Yaskawa INFORM job: pointsmerc3TRJ1.JBI

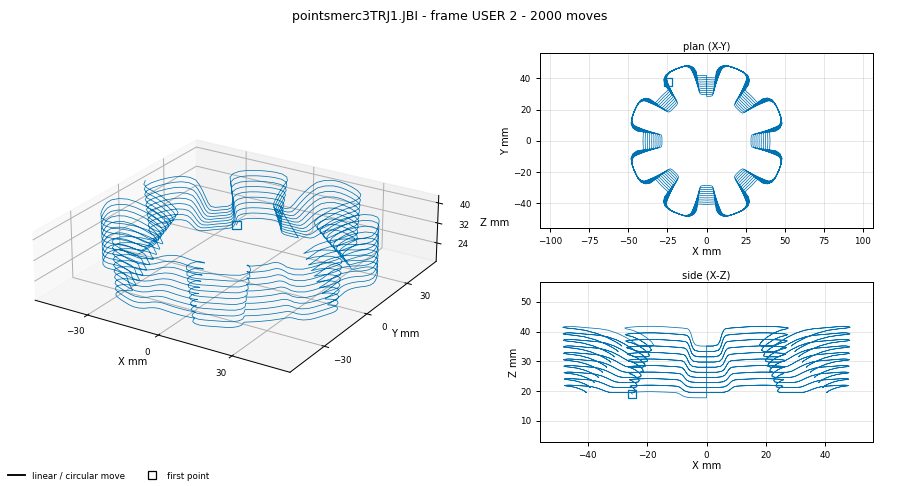
[picture p0: tool path of pointsmerc3TRJ1.JBI in frame USER 2, 2000 of 2000 moves have a stored position in this frame; points joined in program order, loops and branches not executed]
/JOB
//NAME pointsmerc3TRJ1
//POS
///NPOS 2000,0,0,0,0,0
///USER 2
///TOOL 1
///POSTYPE USER
///RECTAN
///RCONF 1,0,0,0,0,0,0,0,0,0,0,0,0,0,0,0,0,0,0,0,0,0,0,0
C00000=-24.917,37.674,19.017,179.9472,0.1674,0.0000
C00001=-25.352,39.110,19.349,-179.2805,-2.8495,0.0000
C00002=-25.558,40.564,19.514,179.7705,-3.0354,0.0000
C00003=-25.030,42.161,19.602,179.1176,-1.5538,0.0000
C00004=-23.802,43.680,19.673,179.0591,-0.8568,0.0000
C00005=-22.056,44.839,19.746,179.9560,-0.0226,0.0000
C00006=-20.124,45.768,19.794,179.9935,-0.0029,0.0000
C00007=-18.133,46.592,19.794,179.9934,-0.0025,0.0000
C00008=-16.110,47.302,19.746,179.9530,-0.0151,0.0000
C00009=-14.056,47.717,19.673,178.7288,-0.0593,0.0000
C00010=-12.113,47.511,19.602,178.2774,0.4749,0.0000
C00011=-10.611,46.755,19.514,177.6906,1.9837,0.0000
C00012=-9.729,45.582,19.349,178.4925,2.5230,0.0000
C00013=-9.020,44.258,19.017,-179.9189,-0.1557,0.0000
C00014=-8.331,43.070,18.587,-176.3263,-5.7834,0.0000
C00015=-7.515,42.203,18.169,-165.2639,-13.0795,0.0000
C00016=-6.279,41.769,17.866,-146.1512,-5.7263,0.0000
C00017=-4.265,41.794,17.745,-142.9346,1.8354,0.0000
C00018=-2.165,41.942,17.740,-142.7693,1.9023,0.0000
C00019=0.000,41.999,17.743,-142.7393,0.0003,0.0000
C00020=0.000,40.651,19.482,-141.7566,0.0003,0.0000
C00021=2.042,40.599,19.478,-141.7861,-1.9186,0.0000
C00022=4.057,40.463,19.484,-141.9733,-1.4629,0.0000
C00023=6.024,40.479,19.630,-146.2958,7.7682,0.0000
C00024=7.200,41.019,19.996,-169.0806,12.4470,0.0000
C00025=7.966,42.055,20.504,-178.0973,3.7099,0.0000
C00026=8.617,43.471,21.031,179.2926,-1.6631,0.0000
C00027=9.290,45.059,21.441,177.9597,-4.2609,0.0000
C00028=10.130,46.493,21.645,176.7689,-3.4833,0.0000
C00029=11.658,47.456,21.754,177.4448,-0.9082,0.0000
C00030=13.694,47.783,21.842,178.3657,0.0207,0.0000
C00031=15.881,47.377,21.932,179.9236,0.0242,0.0000
C00032=18.055,46.622,21.992,179.9901,0.0038,0.0000
C00033=20.200,45.734,21.992,179.9903,0.0044,0.0000
C00034=22.271,44.730,21.932,179.9289,0.0369,0.0000
C00035=24.104,43.471,21.842,178.8296,1.1409,0.0000
C00036=25.313,41.801,21.754,178.8351,2.4489,0.0000
C00037=25.713,40.038,21.645,-179.8172,4.7463,0.0000
C00038=25.293,38.430,21.441,-178.4233,4.4530,0.0000
C00039=24.645,36.832,21.031,-179.3238,1.6761,0.0000
C00040=24.105,35.370,20.504,178.7177,-3.9670,0.0000
C00041=23.913,34.096,19.996,178.7089,-16.4515,0.0000
C00042=24.363,32.883,19.630,-160.4193,-28.9701,0.0000
C00043=25.743,31.481,19.484,-150.0620,-24.6708,0.0000
C00044=27.264,30.151,19.478,-149.5929,-24.4247,0.0000
C00045=28.745,28.745,19.482,-150.8690,-25.9576,0.0000
C00046=30.151,27.264,19.478,-152.2298,-27.4413,0.0000
C00047=31.481,25.743,19.484,-152.0729,-26.9678,0.0000
C00048=32.883,24.363,19.630,-149.5613,-17.0504,0.0000
C00049=34.096,23.913,19.996,-163.5445,1.2382,0.0000
C00050=35.370,24.105,20.504,-176.0321,1.2792,0.0000
C00051=36.832,24.645,21.031,178.3238,-0.6759,0.0000
C00052=38.430,25.293,21.441,175.5453,-1.5719,0.0000
C00053=40.038,25.713,21.645,175.2537,-0.1822,0.0000
C00054=41.801,25.313,21.754,177.5506,1.1638,0.0000
C00055=43.471,24.104,21.842,178.8588,1.1702,0.0000
C00056=44.730,22.271,21.932,179.9631,0.0711,0.0000
C00057=45.734,20.200,21.992,179.9956,0.0097,0.0000
C00058=46.622,18.055,21.992,179.9962,0.0099,0.0000
C00059=47.377,15.881,21.932,179.9758,0.0764,0.0000
C00060=47.783,13.694,21.842,179.9793,1.6343,0.0000
C00061=47.456,11.658,21.754,-179.0909,2.5548,0.0000
C00062=46.493,10.130,21.645,-176.5112,3.2252,0.0000
C00063=45.059,9.290,21.441,-175.7364,2.0346,0.0000
C00064=43.471,8.617,21.031,-178.3368,0.7071,0.0000
C00065=42.055,7.966,20.504,176.2881,-1.8987,0.0000
C00066=41.019,7.200,19.996,167.3309,-10.6597,0.0000
C00067=40.479,6.024,19.630,170.6874,-33.3542,0.0000
C00068=40.463,4.057,19.484,-178.1431,-38.0121,0.0000
C00069=40.599,2.042,19.478,-177.5587,-38.1886,0.0000
C00070=40.651,0.000,19.482,179.9997,-38.2434,0.0000
C00071=40.599,-2.042,19.478,177.5592,-38.1887,0.0000
C00072=40.463,-4.057,19.484,178.1450,-38.0120,0.0000
C00073=40.479,-6.024,19.630,-170.6883,-33.3546,0.0000
C00074=41.019,-7.200,19.996,-167.3309,-10.6597,0.0000
C00075=42.055,-7.966,20.504,-176.2881,-1.8987,0.0000
C00076=43.471,-8.617,21.031,178.3368,0.7071,0.0000
C00077=45.059,-9.290,21.441,175.7364,2.0346,0.0000
C00078=46.493,-10.130,21.645,176.5112,3.2252,0.0000
C00079=47.456,-11.658,21.754,179.0909,2.5548,0.0000
C00080=47.783,-13.694,21.842,-179.9793,1.6343,0.0000
C00081=47.377,-15.881,21.932,-179.9758,0.0764,0.0000
C00082=46.622,-18.055,21.992,-179.9962,0.0099,0.0000
C00083=45.734,-20.200,21.992,-179.9956,0.0097,0.0000
C00084=44.730,-22.271,21.932,-179.9631,0.0711,0.0000
C00085=43.471,-24.104,21.842,-178.8588,1.1702,0.0000
C00086=41.801,-25.313,21.754,-177.5506,1.1638,0.0000
C00087=40.038,-25.713,21.645,-175.2537,-0.1822,0.0000
C00088=38.430,-25.293,21.441,-175.5453,-1.5719,0.0000
C00089=36.832,-24.645,21.031,-178.3238,-0.6759,0.0000
C00090=35.370,-24.105,20.504,176.0321,1.2792,0.0000
C00091=34.096,-23.913,19.996,163.5445,1.2382,0.0000
C00092=32.883,-24.363,19.630,149.5611,-17.0496,0.0000
C00093=31.481,-25.743,19.484,152.0737,-26.9690,0.0000
C00094=30.151,-27.264,19.478,152.2301,-27.4416,0.0000
C00095=28.745,-28.745,19.482,150.8686,-25.9571,0.0000
C00096=27.264,-30.151,19.478,149.5931,-24.4250,0.0000
C00097=25.743,-31.481,19.484,150.0631,-24.6718,0.0000
C00098=24.363,-32.883,19.630,160.4184,-28.9698,0.0000
C00099=23.913,-34.096,19.996,-178.7089,-16.4515,0.0000
C00100=24.105,-35.370,20.504,-178.7177,-3.9670,0.0000
C00101=24.645,-36.832,21.031,179.3238,1.6761,0.0000
C00102=25.293,-38.430,21.441,178.4233,4.4530,0.0000
C00103=25.713,-40.038,21.645,179.8172,4.7463,0.0000
C00104=25.313,-41.801,21.754,-178.8351,2.4489,0.0000
C00105=24.104,-43.471,21.842,-178.8296,1.1409,0.0000
C00106=22.271,-44.730,21.932,-179.9289,0.0369,0.0000
C00107=20.200,-45.734,21.992,-179.9903,0.0044,0.0000
C00108=18.055,-46.622,21.992,-179.9901,0.0038,0.0000
C00109=15.881,-47.377,21.932,-179.9236,0.0242,0.0000
C00110=13.694,-47.783,21.842,-178.3657,0.0207,0.0000
C00111=11.658,-47.456,21.754,-177.4448,-0.9082,0.0000
C00112=10.130,-46.493,21.645,-176.7689,-3.4833,0.0000
C00113=9.290,-45.059,21.441,-177.9597,-4.2609,0.0000
C00114=8.617,-43.471,21.031,-179.2926,-1.6631,0.0000
C00115=7.966,-42.055,20.504,178.0973,3.7099,0.0000
C00116=7.200,-41.019,19.996,169.0806,12.4470,0.0000
C00117=6.024,-40.479,19.630,146.2958,7.7682,0.0000
C00118=4.057,-40.463,19.484,141.9733,-1.4629,0.0000
C00119=2.042,-40.599,19.478,141.7861,-1.9186,0.0000
C00120=0.000,-40.651,19.482,141.7566,0.0003,0.0000
C00121=0.000,-40.651,19.482,141.7566,0.0003,0.0000
C00122=-2.042,-40.599,19.478,141.7861,1.9182,0.0000
C00123=-4.057,-40.463,19.484,141.9735,1.4614,0.0000
C00124=-6.024,-40.479,19.630,146.2954,-7.7675,0.0000
C00125=-7.200,-41.019,19.996,169.0806,-12.4470,0.0000
C00126=-7.966,-42.055,20.504,178.0973,-3.7099,0.0000
C00127=-8.617,-43.471,21.031,-179.2926,1.6631,0.0000
C00128=-9.290,-45.059,21.441,-177.9597,4.2609,0.0000
C00129=-10.130,-46.493,21.645,-176.7689,3.4833,0.0000
C00130=-11.658,-47.456,21.754,-177.4448,0.9082,0.0000
C00131=-13.694,-47.783,21.842,-178.3657,-0.0207,0.0000
C00132=-15.881,-47.377,21.932,-179.9236,-0.0242,0.0000
C00133=-18.055,-46.622,21.992,-179.9901,-0.0038,0.0000
C00134=-20.200,-45.734,21.992,-179.9903,-0.0044,0.0000
C00135=-22.271,-44.730,21.932,-179.9289,-0.0369,0.0000
C00136=-24.104,-43.471,21.842,-178.8296,-1.1409,0.0000
C00137=-25.313,-41.801,21.754,-178.8351,-2.4489,0.0000
C00138=-25.713,-40.038,21.645,179.8172,-4.7463,0.0000
C00139=-25.293,-38.430,21.441,178.4233,-4.4530,0.0000
C00140=-24.645,-36.832,21.031,179.3238,-1.6761,0.0000
C00141=-24.105,-35.370,20.504,-178.7177,3.9670,0.0000
C00142=-23.913,-34.096,19.996,-178.7089,16.4515,0.0000
C00143=-24.363,-32.883,19.630,160.4193,28.9701,0.0000
C00144=-25.743,-31.481,19.484,150.0620,24.6708,0.0000
C00145=-27.264,-30.151,19.478,149.5929,24.4247,0.0000
C00146=-28.745,-28.745,19.482,150.8690,25.9576,0.0000
C00147=-30.151,-27.264,19.478,152.2298,27.4413,0.0000
C00148=-31.481,-25.743,19.484,152.0729,26.9678,0.0000
C00149=-32.883,-24.363,19.630,149.5613,17.0504,0.0000
C00150=-34.096,-23.913,19.996,163.5445,-1.2382,0.0000
C00151=-35.370,-24.105,20.504,176.0321,-1.2792,0.0000
C00152=-36.832,-24.645,21.031,-178.3238,0.6759,0.0000
C00153=-38.430,-25.293,21.441,-175.5453,1.5719,0.0000
C00154=-40.038,-25.713,21.645,-175.2537,0.1822,0.0000
C00155=-41.801,-25.313,21.754,-177.5506,-1.1638,0.0000
C00156=-43.471,-24.104,21.842,-178.8588,-1.1702,0.0000
C00157=-44.730,-22.271,21.932,-179.9631,-0.0711,0.0000
C00158=-45.734,-20.200,21.992,-179.9956,-0.0097,0.0000
C00159=-46.622,-18.055,21.992,-179.9962,-0.0099,0.0000
C00160=-47.377,-15.881,21.932,-179.9758,-0.0764,0.0000
C00161=-47.783,-13.694,21.842,-179.9793,-1.6343,0.0000
C00162=-47.456,-11.658,21.754,179.0909,-2.5548,0.0000
C00163=-46.493,-10.130,21.645,176.5112,-3.2252,0.0000
C00164=-45.059,-9.290,21.441,175.7364,-2.0346,0.0000
C00165=-43.471,-8.617,21.031,178.3368,-0.7071,0.0000
C00166=-42.055,-7.966,20.504,-176.2881,1.8987,0.0000
C00167=-41.019,-7.200,19.996,-167.3309,10.6597,0.0000
C00168=-40.479,-6.024,19.630,-170.6874,33.3542,0.0000
C00169=-40.463,-4.057,19.484,178.1431,38.0121,0.0000
C00170=-40.599,-2.042,19.478,177.5587,38.1886,0.0000
C00171=-40.651,0.000,19.482,-179.9997,38.2434,0.0000
C00172=-40.599,2.042,19.478,-177.5592,38.1887,0.0000
C00173=-40.463,4.057,19.484,-178.1450,38.0120,0.0000
C00174=-40.479,6.024,19.630,170.6883,33.3546,0.0000
C00175=-41.019,7.200,19.996,167.3309,10.6597,0.0000
C00176=-42.055,7.966,20.504,176.2881,1.8987,0.0000
C00177=-43.471,8.617,21.031,-178.3368,-0.7071,0.0000
C00178=-45.059,9.290,21.441,-175.7364,-2.0346,0.0000
C00179=-46.493,10.130,21.645,-176.5112,-3.2252,0.0000
C00180=-47.456,11.658,21.754,-179.0909,-2.5548,0.0000
C00181=-47.783,13.694,21.842,179.9793,-1.6343,0.0000
C00182=-47.377,15.881,21.932,179.9758,-0.0764,0.0000
C00183=-46.622,18.055,21.992,179.9962,-0.0099,0.0000
C00184=-45.734,20.200,21.992,179.9956,-0.0097,0.0000
C00185=-44.730,22.271,21.932,179.9631,-0.0711,0.0000
C00186=-43.471,24.104,21.842,178.8588,-1.1702,0.0000
C00187=-41.801,25.313,21.754,177.5506,-1.1638,0.0000
C00188=-40.038,25.713,21.645,175.2537,0.1822,0.0000
C00189=-38.430,25.293,21.441,175.5453,1.5719,0.0000
C00190=-36.832,24.645,21.031,178.3238,0.6759,0.0000
C00191=-35.370,24.105,20.504,-176.0321,-1.2792,0.0000
C00192=-34.096,23.913,19.996,-163.5445,-1.2382,0.0000
C00193=-32.883,24.363,19.630,-149.5611,17.0496,0.0000
C00194=-31.481,25.743,19.484,-152.0737,26.9690,0.0000
C00195=-30.151,27.264,19.478,-152.2301,27.4416,0.0000
C00196=-28.745,28.745,19.482,-150.8686,25.9571,0.0000
C00197=-27.264,30.151,19.478,-149.5931,24.4250,0.0000
C00198=-25.743,31.481,19.484,-150.0631,24.6718,0.0000
C00199=-24.363,32.883,19.630,-160.4184,28.9698,0.0000
C00200=-23.913,34.096,19.996,178.7089,16.4515,0.0000
C00201=-24.105,35.370,20.504,178.7177,3.9670,0.0000
C00202=-24.645,36.832,21.031,-179.3238,-1.6761,0.0000
C00203=-25.293,38.430,21.441,-178.4233,-4.4530,0.0000
C00204=-25.713,40.038,21.645,-179.8172,-4.7463,0.0000
C00205=-25.313,41.801,21.754,178.8351,-2.4489,0.0000
C00206=-24.104,43.471,21.842,178.8296,-1.1409,0.0000
C00207=-22.271,44.730,21.932,179.9289,-0.0369,0.0000
C00208=-20.200,45.734,21.992,179.9903,-0.0044,0.0000
C00209=-18.055,46.622,21.992,179.9901,-0.0038,0.0000
C00210=-15.881,47.377,21.932,179.9236,-0.0242,0.0000
C00211=-13.694,47.783,21.842,178.3657,-0.0207,0.0000
C00212=-11.658,47.456,21.754,177.4448,0.9082,0.0000
C00213=-10.130,46.493,21.645,176.7689,3.4833,0.0000
C00214=-9.290,45.059,21.441,177.9597,4.2609,0.0000
C00215=-8.617,43.471,21.031,179.2926,1.6631,0.0000
C00216=-7.966,42.055,20.504,-178.0973,-3.7099,0.0000
C00217=-7.200,41.019,19.996,-169.0806,-12.4470,0.0000
C00218=-6.024,40.479,19.630,-146.2954,-7.7675,0.0000
C00219=-4.057,40.463,19.484,-141.9735,1.4614,0.0000
C00220=-2.042,40.599,19.478,-141.7861,1.9182,0.0000
C00221=0.000,40.651,19.482,-141.7566,0.0003,0.0000
C00222=0.000,39.279,21.202,-141.1100,0.0002,0.0000
C00223=1.916,39.231,21.197,-141.1387,-1.9150,0.0000
C00224=3.846,39.107,21.204,-141.3582,-1.0288,0.0000
C00225=5.765,39.166,21.375,-147.0450,9.7425,0.0000
C00226=6.881,39.812,21.808,-172.3813,10.8619,0.0000
C00227=7.594,41.021,22.410,-179.2636,1.7324,0.0000
C00228=8.207,42.669,23.038,178.8678,-3.1758,0.0000
C00229=8.843,44.528,23.528,177.7717,-5.6527,0.0000
C00230=9.641,46.227,23.773,176.2825,-4.8520,0.0000
C00231=11.196,47.401,23.904,176.7678,-1.3919,0.0000
C00232=13.327,47.850,24.010,178.0518,-0.0356,0.0000
C00233=15.648,47.454,24.119,179.8977,0.0319,0.0000
C00234=17.976,46.653,24.190,179.9872,0.0049,0.0000
C00235=20.278,45.699,24.190,179.9875,0.0056,0.0000
C00236=22.491,44.620,24.119,179.9051,0.0498,0.0000
C00237=24.412,43.258,24.010,178.6473,1.4026,0.0000
C00238=25.601,41.434,23.904,178.6983,3.2695,0.0000
C00239=25.871,39.504,23.773,-179.1860,6.0555,0.0000
C00240=25.233,37.739,23.528,-177.5648,5.5670,0.0000
C00241=24.369,35.974,23.038,-178.5526,3.0452,0.0000
C00242=23.637,34.376,22.410,179.2953,-1.7456,0.0000
C00243=23.286,33.017,21.808,177.5775,-13.0215,0.0000
C00244=23.618,31.771,21.375,-162.5821,-29.9181,0.0000
C00245=24.933,30.373,21.204,-149.8186,-25.3906,0.0000
C00246=26.385,29.096,21.197,-149.0304,-24.8212,0.0000
C00247=27.774,27.774,21.202,-150.3014,-26.3558,0.0000
C00248=29.096,26.385,21.197,-151.6568,-27.8426,0.0000
C00249=30.373,24.933,21.204,-151.2294,-27.0106,0.0000
C00250=31.771,23.618,21.375,-148.9059,-15.0382,0.0000
C00251=33.017,23.286,21.808,-166.9673,2.3601,0.0000
C00252=34.376,23.637,22.410,-178.2543,0.7044,0.0000
C00253=35.974,24.369,23.038,176.9538,-1.4453,0.0000
C00254=37.739,25.233,23.528,174.4280,-2.4237,0.0000
C00255=39.504,25.871,23.773,173.9439,-0.8094,0.0000
C00256=41.434,25.601,23.904,176.7297,1.2996,0.0000
C00257=43.258,24.412,24.010,178.5970,1.3523,0.0000
C00258=44.620,22.491,24.119,179.9502,0.0949,0.0000
C00259=45.699,20.278,24.190,179.9944,0.0125,0.0000
C00260=46.653,17.976,24.190,179.9951,0.0128,0.0000
C00261=47.454,15.648,24.119,179.9681,0.1023,0.0000
C00262=47.850,13.327,24.010,-179.9644,1.9482,0.0000
C00263=47.401,11.196,23.904,-178.6059,3.2312,0.0000
C00264=46.227,9.641,23.773,-175.1378,3.7041,0.0000
C00265=44.528,8.843,23.528,-174.3430,2.2175,0.0000
C00266=42.669,8.207,23.038,-176.8236,1.1304,0.0000
C00267=41.021,7.594,22.410,178.2674,-0.7361,0.0000
C00268=39.812,6.881,21.808,169.0437,-7.4814,0.0000
C00269=39.166,5.765,21.375,168.4358,-32.4210,0.0000
C00270=39.107,3.846,21.204,-178.6830,-38.6345,0.0000
C00271=39.231,1.916,21.197,-177.5412,-38.8355,0.0000
C00272=39.279,0.000,21.202,179.9998,-38.8900,0.0000
C00273=39.231,-1.916,21.197,177.5416,-38.8356,0.0000
C00274=39.107,-3.847,21.204,178.6850,-38.6342,0.0000
C00275=39.166,-5.765,21.375,-168.4365,-32.4215,0.0000
C00276=39.812,-6.881,21.808,-169.0437,-7.4814,0.0000
C00277=41.021,-7.594,22.410,-178.2674,-0.7361,0.0000
C00278=42.669,-8.207,23.038,176.8236,1.1304,0.0000
C00279=44.528,-8.843,23.528,174.3430,2.2175,0.0000
C00280=46.227,-9.641,23.773,175.1378,3.7041,0.0000
C00281=47.401,-11.196,23.904,178.6059,3.2312,0.0000
C00282=47.850,-13.327,24.010,179.9644,1.9482,0.0000
C00283=47.454,-15.648,24.119,-179.9681,0.1023,0.0000
C00284=46.653,-17.976,24.190,-179.9951,0.0128,0.0000
C00285=45.699,-20.278,24.190,-179.9944,0.0125,0.0000
C00286=44.620,-22.491,24.119,-179.9502,0.0949,0.0000
C00287=43.258,-24.412,24.010,-178.5970,1.3523,0.0000
C00288=41.434,-25.601,23.904,-176.7297,1.2996,0.0000
C00289=39.504,-25.871,23.773,-173.9439,-0.8094,0.0000
C00290=37.739,-25.233,23.528,-174.4280,-2.4237,0.0000
C00291=35.974,-24.369,23.038,-176.9538,-1.4453,0.0000
C00292=34.376,-23.637,22.410,178.2543,0.7044,0.0000
C00293=33.017,-23.286,21.808,166.9673,2.3601,0.0000
C00294=31.771,-23.618,21.375,148.9058,-15.0373,0.0000
C00295=30.373,-24.933,21.204,151.2304,-27.0120,0.0000
C00296=29.096,-26.385,21.197,151.6570,-27.8428,0.0000
C00297=27.774,-27.774,21.202,150.3012,-26.3555,0.0000
C00298=26.385,-29.096,21.197,149.0306,-24.8215,0.0000
C00299=24.933,-30.373,21.204,149.8199,-25.3917,0.0000
C00300=23.618,-31.771,21.375,162.5812,-29.9179,0.0000
C00301=23.286,-33.017,21.808,-177.5775,-13.0215,0.0000
C00302=23.637,-34.376,22.410,-179.2953,-1.7456,0.0000
C00303=24.369,-35.974,23.038,178.5526,3.0452,0.0000
C00304=25.233,-37.739,23.528,177.5648,5.5670,0.0000
C00305=25.871,-39.504,23.773,179.1860,6.0555,0.0000
C00306=25.601,-41.434,23.904,-178.6983,3.2695,0.0000
C00307=24.412,-43.258,24.010,-178.6473,1.4026,0.0000
C00308=22.491,-44.620,24.119,-179.9051,0.0498,0.0000
C00309=20.278,-45.699,24.190,-179.9875,0.0056,0.0000
C00310=17.976,-46.653,24.190,-179.9872,0.0049,0.0000
C00311=15.648,-47.454,24.119,-179.8977,0.0319,0.0000
C00312=13.327,-47.850,24.010,-178.0518,-0.0356,0.0000
C00313=11.196,-47.401,23.904,-176.7678,-1.3919,0.0000
C00314=9.641,-46.227,23.773,-176.2825,-4.8520,0.0000
C00315=8.843,-44.528,23.528,-177.7717,-5.6527,0.0000
C00316=8.207,-42.669,23.038,-178.8678,-3.1758,0.0000
C00317=7.594,-41.021,22.410,179.2636,1.7324,0.0000
C00318=6.881,-39.812,21.808,172.3813,10.8619,0.0000
C00319=5.765,-39.166,21.375,147.0450,9.7425,0.0000
C00320=3.846,-39.107,21.204,141.3582,-1.0288,0.0000
C00321=1.916,-39.231,21.197,141.1387,-1.9150,0.0000
C00322=0.000,-39.279,21.202,141.1100,0.0002,0.0000
C00323=0.000,-39.279,21.202,141.1100,0.0002,0.0000
C00324=-1.916,-39.231,21.197,141.1386,1.9147,0.0000
C00325=-3.847,-39.107,21.204,141.3584,1.0272,0.0000
C00326=-5.765,-39.166,21.375,147.0445,-9.7418,0.0000
C00327=-6.881,-39.812,21.808,172.3813,-10.8619,0.0000
C00328=-7.594,-41.021,22.410,179.2636,-1.7324,0.0000
C00329=-8.207,-42.669,23.038,-178.8678,3.1758,0.0000
C00330=-8.843,-44.528,23.528,-177.7717,5.6527,0.0000
C00331=-9.641,-46.227,23.773,-176.2825,4.8520,0.0000
C00332=-11.196,-47.401,23.904,-176.7678,1.3919,0.0000
C00333=-13.327,-47.850,24.010,-178.0518,0.0356,0.0000
C00334=-15.648,-47.454,24.119,-179.8977,-0.0319,0.0000
C00335=-17.976,-46.653,24.190,-179.9872,-0.0049,0.0000
C00336=-20.278,-45.699,24.190,-179.9875,-0.0056,0.0000
C00337=-22.491,-44.620,24.119,-179.9051,-0.0498,0.0000
C00338=-24.412,-43.258,24.010,-178.6473,-1.4026,0.0000
C00339=-25.601,-41.434,23.904,-178.6983,-3.2695,0.0000
C00340=-25.871,-39.504,23.773,179.1860,-6.0555,0.0000
C00341=-25.233,-37.739,23.528,177.5648,-5.5670,0.0000
C00342=-24.369,-35.974,23.038,178.5526,-3.0452,0.0000
C00343=-23.637,-34.376,22.410,-179.2953,1.7456,0.0000
C00344=-23.286,-33.017,21.808,-177.5775,13.0215,0.0000
C00345=-23.618,-31.771,21.375,162.5821,29.9181,0.0000
C00346=-24.933,-30.373,21.204,149.8186,25.3906,0.0000
C00347=-26.385,-29.096,21.197,149.0304,24.8212,0.0000
C00348=-27.774,-27.774,21.202,150.3014,26.3558,0.0000
C00349=-29.096,-26.385,21.197,151.6568,27.8426,0.0000
C00350=-30.373,-24.933,21.204,151.2294,27.0106,0.0000
C00351=-31.771,-23.618,21.375,148.9059,15.0382,0.0000
C00352=-33.017,-23.286,21.808,166.9673,-2.3601,0.0000
C00353=-34.376,-23.637,22.410,178.2543,-0.7044,0.0000
C00354=-35.974,-24.369,23.038,-176.9538,1.4453,0.0000
C00355=-37.739,-25.233,23.528,-174.4280,2.4237,0.0000
C00356=-39.504,-25.871,23.773,-173.9439,0.8094,0.0000
C00357=-41.434,-25.601,23.904,-176.7297,-1.2996,0.0000
C00358=-43.258,-24.412,24.010,-178.5970,-1.3523,0.0000
C00359=-44.620,-22.491,24.119,-179.9502,-0.0949,0.0000
C00360=-45.699,-20.278,24.190,-179.9944,-0.0125,0.0000
C00361=-46.653,-17.976,24.190,-179.9951,-0.0128,0.0000
C00362=-47.454,-15.648,24.119,-179.9681,-0.1023,0.0000
C00363=-47.850,-13.327,24.010,179.9644,-1.9482,0.0000
C00364=-47.401,-11.196,23.904,178.6059,-3.2312,0.0000
C00365=-46.227,-9.641,23.773,175.1378,-3.7041,0.0000
C00366=-44.528,-8.843,23.528,174.3430,-2.2175,0.0000
C00367=-42.669,-8.207,23.038,176.8236,-1.1304,0.0000
C00368=-41.021,-7.594,22.410,-178.2674,0.7361,0.0000
C00369=-39.812,-6.881,21.808,-169.0437,7.4814,0.0000
C00370=-39.166,-5.765,21.375,-168.4358,32.4210,0.0000
C00371=-39.107,-3.846,21.204,178.6830,38.6345,0.0000
C00372=-39.231,-1.916,21.197,177.5412,38.8355,0.0000
C00373=-39.279,0.000,21.202,-179.9998,38.8900,0.0000
C00374=-39.231,1.916,21.197,-177.5416,38.8356,0.0000
C00375=-39.107,3.847,21.204,-178.6850,38.6342,0.0000
C00376=-39.166,5.765,21.375,168.4365,32.4215,0.0000
C00377=-39.812,6.881,21.808,169.0437,7.4814,0.0000
C00378=-41.021,7.594,22.410,178.2674,0.7361,0.0000
C00379=-42.669,8.207,23.038,-176.8236,-1.1304,0.0000
C00380=-44.528,8.843,23.528,-174.3430,-2.2175,0.0000
C00381=-46.227,9.641,23.773,-175.1378,-3.7041,0.0000
C00382=-47.401,11.196,23.904,-178.6059,-3.2312,0.0000
C00383=-47.850,13.327,24.010,-179.9644,-1.9482,0.0000
C00384=-47.454,15.648,24.119,179.9681,-0.1023,0.0000
C00385=-46.653,17.976,24.190,179.9951,-0.0128,0.0000
C00386=-45.699,20.278,24.190,179.9944,-0.0125,0.0000
C00387=-44.620,22.491,24.119,179.9502,-0.0949,0.0000
C00388=-43.258,24.412,24.010,178.5970,-1.3523,0.0000
C00389=-41.434,25.601,23.904,176.7297,-1.2996,0.0000
C00390=-39.504,25.871,23.773,173.9439,0.8094,0.0000
C00391=-37.739,25.233,23.528,174.4280,2.4237,0.0000
C00392=-35.974,24.369,23.038,176.9538,1.4453,0.0000
C00393=-34.376,23.637,22.410,-178.2543,-0.7044,0.0000
C00394=-33.017,23.286,21.808,-166.9673,-2.3601,0.0000
C00395=-31.771,23.618,21.375,-148.9058,15.0373,0.0000
C00396=-30.373,24.933,21.204,-151.2304,27.0120,0.0000
C00397=-29.096,26.385,21.197,-151.6570,27.8428,0.0000
C00398=-27.774,27.774,21.202,-150.3012,26.3555,0.0000
C00399=-26.385,29.096,21.197,-149.0306,24.8215,0.0000
C00400=-24.933,30.373,21.204,-149.8199,25.3917,0.0000
C00401=-23.618,31.771,21.375,-162.5812,29.9179,0.0000
C00402=-23.286,33.017,21.808,177.5775,13.0215,0.0000
C00403=-23.637,34.376,22.410,179.2953,1.7456,0.0000
C00404=-24.369,35.974,23.038,-178.5526,-3.0452,0.0000
C00405=-25.233,37.739,23.528,-177.5648,-5.5670,0.0000
C00406=-25.871,39.504,23.773,-179.1860,-6.0555,0.0000
C00407=-25.601,41.434,23.904,178.6983,-3.2695,0.0000
C00408=-24.412,43.258,24.010,178.6473,-1.4026,0.0000
C00409=-22.491,44.620,24.119,179.9051,-0.0498,0.0000
C00410=-20.278,45.699,24.190,179.9875,-0.0056,0.0000
C00411=-17.976,46.653,24.190,179.9872,-0.0049,0.0000
C00412=-15.648,47.454,24.119,179.8977,-0.0319,0.0000
C00413=-13.327,47.850,24.010,178.0518,0.0356,0.0000
C00414=-11.196,47.401,23.904,176.7678,1.3919,0.0000
C00415=-9.641,46.227,23.773,176.2825,4.8520,0.0000
C00416=-8.843,44.528,23.528,177.7717,5.6527,0.0000
C00417=-8.207,42.669,23.038,178.8678,3.1758,0.0000
C00418=-7.594,41.021,22.410,-179.2636,-1.7324,0.0000
C00419=-6.881,39.812,21.808,-172.3813,-10.8619,0.0000
C00420=-5.765,39.166,21.375,-147.0445,-9.7418,0.0000
C00421=-3.847,39.107,21.204,-141.3584,1.0272,0.0000
C00422=-1.916,39.231,21.197,-141.1386,1.9147,0.0000
C00423=0.000,39.279,21.202,-141.1100,0.0002,0.0000
C00424=0.000,37.892,22.909,-140.7729,0.0001,0.0000
C00425=1.790,37.849,22.904,-140.8005,-1.8934,0.0000
C00426=3.633,37.737,22.912,-141.0647,-0.5438,0.0000
C00427=5.504,37.838,23.110,-148.3550,11.5394,0.0000
C00428=6.557,38.594,23.612,-174.9776,8.7701,0.0000
C00429=7.219,39.979,24.311,-179.9995,0.0014,0.0000
C00430=7.794,41.862,25.043,178.6707,-4.3586,0.0000
C00431=8.395,43.994,25.615,177.7869,-6.6761,0.0000
C00432=9.151,45.960,25.902,176.1277,-5.9542,0.0000
C00433=10.734,47.345,26.054,176.2738,-1.8650,0.0000
C00434=12.959,47.917,26.178,177.8036,-0.1012,0.0000
C00435=15.415,47.531,26.305,179.8764,0.0380,0.0000
C00436=17.897,46.683,26.389,179.9849,0.0057,0.0000
C00437=20.355,45.665,26.389,179.9853,0.0067,0.0000
C00438=22.710,44.510,26.305,179.8857,0.0605,0.0000
C00439=24.719,43.046,26.178,178.5181,1.6245,0.0000
C00440=25.888,41.068,26.054,178.6837,3.9532,0.0000
C00441=26.028,38.969,25.902,-178.5075,6.9409,0.0000
C00442=25.172,37.045,25.615,-176.8232,6.2765,0.0000
C00443=24.090,35.112,25.043,-177.8523,4.0195,0.0000
C00444=23.165,33.374,24.311,179.9993,-0.0014,0.0000
C00445=22.654,31.927,23.612,177.2881,-9.7292,0.0000
C00446=22.864,30.647,23.110,-165.0937,-30.3273,0.0000
C00447=24.115,29.253,22.912,-149.8901,-25.9537,0.0000
C00448=25.498,28.029,22.904,-148.7483,-25.0431,0.0000
C00449=26.793,26.793,22.909,-150.0040,-26.5624,0.0000
C00450=28.029,25.498,22.904,-151.3420,-28.0359,0.0000
C00451=29.253,24.115,22.912,-150.6345,-26.8106,0.0000
C00452=30.647,22.864,23.110,-148.8108,-12.8294,0.0000
C00453=31.927,22.654,23.612,-170.2601,2.6728,0.0000
C00454=33.374,23.165,24.311,-179.9986,0.0007,0.0000
C00455=35.112,24.090,25.043,175.9777,-2.1424,0.0000
C00456=37.045,25.172,25.615,173.7139,-3.1578,0.0000
C00457=38.969,26.028,25.902,173.0567,-1.4816,0.0000
C00458=41.068,25.888,26.054,176.0457,1.3131,0.0000
C00459=43.046,24.719,26.178,178.3750,1.4813,0.0000
C00460=44.510,22.710,26.305,179.9395,0.1143,0.0000
C00461=45.665,20.355,26.389,179.9933,0.0147,0.0000
C00462=46.683,17.897,26.389,179.9943,0.0151,0.0000
C00463=47.531,15.415,26.305,179.9620,0.1236,0.0000
C00464=47.917,12.959,26.178,-179.8987,2.1964,0.0000
C00465=47.345,10.734,26.054,-178.1310,3.7242,0.0000
C00466=45.960,9.151,25.902,-174.0323,3.8514,0.0000
C00467=43.994,8.395,25.615,-173.3189,2.1980,0.0000
C00468=41.862,7.794,25.043,-175.6402,1.3254,0.0000
C00469=39.979,7.219,24.311,179.9986,-0.0005,0.0000
C00470=38.594,6.557,23.612,171.1966,-4.9635,0.0000
C00471=37.838,5.504,23.110,166.5136,-30.9339,0.0000
C00472=37.737,3.633,22.912,-179.3009,-38.9332,0.0000
C00473=37.849,1.790,22.904,-177.5573,-39.1740,0.0000
C00474=37.892,0.000,22.909,179.9999,-39.2271,0.0000
C00475=37.849,-1.790,22.904,177.5576,-39.1740,0.0000
C00476=37.737,-3.633,22.912,179.3032,-38.9330,0.0000
C00477=37.838,-5.504,23.110,-166.5142,-30.9345,0.0000
C00478=38.594,-6.557,23.612,-171.1966,-4.9635,0.0000
C00479=39.979,-7.219,24.311,-179.9986,-0.0005,0.0000
C00480=41.862,-7.794,25.043,175.6402,1.3254,0.0000
C00481=43.994,-8.395,25.615,173.3189,2.1980,0.0000
C00482=45.960,-9.151,25.902,174.0323,3.8514,0.0000
C00483=47.345,-10.734,26.054,178.1310,3.7242,0.0000
C00484=47.917,-12.959,26.178,179.8987,2.1964,0.0000
C00485=47.531,-15.415,26.305,-179.9620,0.1236,0.0000
C00486=46.683,-17.897,26.389,-179.9943,0.0151,0.0000
C00487=45.665,-20.355,26.389,-179.9933,0.0147,0.0000
C00488=44.510,-22.710,26.305,-179.9395,0.1143,0.0000
C00489=43.046,-24.719,26.178,-178.3750,1.4813,0.0000
C00490=41.068,-25.888,26.054,-176.0457,1.3131,0.0000
C00491=38.969,-26.028,25.902,-173.0567,-1.4816,0.0000
C00492=37.045,-25.172,25.615,-173.7139,-3.1578,0.0000
C00493=35.112,-24.090,25.043,-175.9777,-2.1424,0.0000
C00494=33.374,-23.165,24.311,179.9986,0.0007,0.0000
C00495=31.927,-22.654,23.612,170.2601,2.6728,0.0000
C00496=30.647,-22.864,23.110,148.8108,-12.8287,0.0000
C00497=29.253,-24.115,22.912,150.6355,-26.8122,0.0000
C00498=28.029,-25.498,22.904,151.3422,-28.0360,0.0000
C00499=26.793,-26.793,22.909,150.0039,-26.5623,0.0000
C00500=25.498,-28.029,22.904,148.7484,-25.0433,0.0000
C00501=24.115,-29.253,22.912,149.8915,-25.9549,0.0000
C00502=22.864,-30.647,23.110,165.0929,-30.3272,0.0000
C00503=22.654,-31.927,23.612,-177.2881,-9.7292,0.0000
C00504=23.165,-33.374,24.311,-179.9993,-0.0014,0.0000
C00505=24.090,-35.112,25.043,177.8523,4.0195,0.0000
C00506=25.172,-37.045,25.615,176.8232,6.2765,0.0000
C00507=26.028,-38.969,25.902,178.5075,6.9409,0.0000
C00508=25.888,-41.068,26.054,-178.6837,3.9532,0.0000
C00509=24.719,-43.046,26.178,-178.5181,1.6245,0.0000
C00510=22.710,-44.510,26.305,-179.8857,0.0605,0.0000
C00511=20.355,-45.665,26.389,-179.9853,0.0067,0.0000
C00512=17.897,-46.683,26.389,-179.9849,0.0057,0.0000
C00513=15.415,-47.531,26.305,-179.8764,0.0380,0.0000
C00514=12.959,-47.917,26.178,-177.8036,-0.1012,0.0000
C00515=10.734,-47.345,26.054,-176.2738,-1.8650,0.0000
C00516=9.151,-45.960,25.902,-176.1277,-5.9542,0.0000
C00517=8.395,-43.994,25.615,-177.7869,-6.6761,0.0000
C00518=7.794,-41.862,25.043,-178.6707,-4.3586,0.0000
C00519=7.219,-39.979,24.311,179.9995,0.0014,0.0000
C00520=6.557,-38.594,23.612,174.9776,8.7701,0.0000
C00521=5.504,-37.838,23.110,148.3550,11.5394,0.0000
C00522=3.633,-37.737,22.912,141.0647,-0.5438,0.0000
C00523=1.790,-37.849,22.904,140.8005,-1.8934,0.0000
C00524=0.000,-37.892,22.909,140.7729,0.0001,0.0000
C00525=0.000,-37.892,22.909,140.7729,0.0001,0.0000
C00526=-1.790,-37.849,22.904,140.8005,1.8932,0.0000
C00527=-3.633,-37.737,22.912,141.0650,0.5420,0.0000
C00528=-5.504,-37.838,23.110,148.3545,-11.5388,0.0000
C00529=-6.557,-38.594,23.612,174.9776,-8.7701,0.0000
C00530=-7.219,-39.979,24.311,179.9995,-0.0014,0.0000
C00531=-7.794,-41.862,25.043,-178.6707,4.3586,0.0000
C00532=-8.395,-43.994,25.615,-177.7869,6.6761,0.0000
C00533=-9.151,-45.960,25.902,-176.1277,5.9542,0.0000
C00534=-10.734,-47.345,26.054,-176.2738,1.8650,0.0000
C00535=-12.959,-47.917,26.178,-177.8036,0.1012,0.0000
C00536=-15.415,-47.531,26.305,-179.8764,-0.0380,0.0000
C00537=-17.897,-46.683,26.389,-179.9849,-0.0057,0.0000
C00538=-20.355,-45.665,26.389,-179.9853,-0.0067,0.0000
C00539=-22.710,-44.510,26.305,-179.8857,-0.0605,0.0000
C00540=-24.719,-43.046,26.178,-178.5181,-1.6245,0.0000
C00541=-25.888,-41.068,26.054,-178.6837,-3.9532,0.0000
C00542=-26.028,-38.969,25.902,178.5075,-6.9409,0.0000
C00543=-25.172,-37.045,25.615,176.8232,-6.2765,0.0000
C00544=-24.090,-35.112,25.043,177.8523,-4.0195,0.0000
C00545=-23.165,-33.374,24.311,-179.9993,0.0014,0.0000
C00546=-22.654,-31.927,23.612,-177.2881,9.7292,0.0000
C00547=-22.864,-30.647,23.110,165.0937,30.3273,0.0000
C00548=-24.115,-29.253,22.912,149.8901,25.9537,0.0000
C00549=-25.498,-28.029,22.904,148.7483,25.0431,0.0000
C00550=-26.793,-26.793,22.909,150.0040,26.5624,0.0000
C00551=-28.029,-25.498,22.904,151.3420,28.0359,0.0000
C00552=-29.253,-24.115,22.912,150.6345,26.8106,0.0000
C00553=-30.647,-22.864,23.110,148.8108,12.8294,0.0000
C00554=-31.927,-22.654,23.612,170.2601,-2.6728,0.0000
C00555=-33.374,-23.165,24.311,179.9986,-0.0007,0.0000
C00556=-35.112,-24.090,25.043,-175.9777,2.1424,0.0000
C00557=-37.045,-25.172,25.615,-173.7139,3.1578,0.0000
C00558=-38.969,-26.028,25.902,-173.0567,1.4816,0.0000
C00559=-41.068,-25.888,26.054,-176.0457,-1.3131,0.0000
C00560=-43.046,-24.719,26.178,-178.3750,-1.4813,0.0000
C00561=-44.510,-22.710,26.305,-179.9395,-0.1143,0.0000
C00562=-45.665,-20.355,26.389,-179.9933,-0.0147,0.0000
C00563=-46.683,-17.897,26.389,-179.9943,-0.0151,0.0000
C00564=-47.531,-15.415,26.305,-179.9620,-0.1236,0.0000
C00565=-47.917,-12.959,26.178,179.8987,-2.1964,0.0000
C00566=-47.345,-10.734,26.054,178.1310,-3.7242,0.0000
C00567=-45.960,-9.151,25.902,174.0323,-3.8514,0.0000
C00568=-43.994,-8.395,25.615,173.3189,-2.1980,0.0000
C00569=-41.862,-7.794,25.043,175.6402,-1.3254,0.0000
C00570=-39.979,-7.219,24.311,-179.9986,0.0005,0.0000
C00571=-38.594,-6.557,23.612,-171.1966,4.9635,0.0000
C00572=-37.838,-5.504,23.110,-166.5136,30.9339,0.0000
C00573=-37.737,-3.633,22.912,179.3009,38.9332,0.0000
C00574=-37.849,-1.790,22.904,177.5573,39.1740,0.0000
C00575=-37.892,0.000,22.909,-179.9999,39.2271,0.0000
C00576=-37.849,1.790,22.904,-177.5576,39.1740,0.0000
C00577=-37.737,3.633,22.912,-179.3032,38.9330,0.0000
C00578=-37.838,5.504,23.110,166.5142,30.9345,0.0000
C00579=-38.594,6.557,23.612,171.1966,4.9635,0.0000
C00580=-39.979,7.219,24.311,179.9986,0.0005,0.0000
C00581=-41.862,7.794,25.043,-175.6402,-1.3254,0.0000
C00582=-43.994,8.395,25.615,-173.3189,-2.1980,0.0000
C00583=-45.960,9.151,25.902,-174.0323,-3.8514,0.0000
C00584=-47.345,10.734,26.054,-178.1310,-3.7242,0.0000
C00585=-47.917,12.959,26.178,-179.8987,-2.1964,0.0000
C00586=-47.531,15.415,26.305,179.9620,-0.1236,0.0000
C00587=-46.683,17.897,26.389,179.9943,-0.0151,0.0000
C00588=-45.665,20.355,26.389,179.9933,-0.0147,0.0000
C00589=-44.510,22.710,26.305,179.9395,-0.1143,0.0000
C00590=-43.046,24.719,26.178,178.3750,-1.4813,0.0000
C00591=-41.068,25.888,26.054,176.0457,-1.3131,0.0000
C00592=-38.969,26.028,25.902,173.0567,1.4816,0.0000
C00593=-37.045,25.172,25.615,173.7139,3.1578,0.0000
C00594=-35.112,24.090,25.043,175.9777,2.1424,0.0000
C00595=-33.374,23.165,24.311,-179.9986,-0.0007,0.0000
C00596=-31.927,22.654,23.612,-170.2601,-2.6728,0.0000
C00597=-30.647,22.864,23.110,-148.8108,12.8287,0.0000
C00598=-29.253,24.115,22.912,-150.6355,26.8122,0.0000
C00599=-28.029,25.498,22.904,-151.3422,28.0360,0.0000
C00600=-26.793,26.793,22.909,-150.0039,26.5623,0.0000
C00601=-25.498,28.029,22.904,-148.7484,25.0433,0.0000
C00602=-24.115,29.253,22.912,-149.8915,25.9549,0.0000
C00603=-22.864,30.647,23.110,-165.0929,30.3272,0.0000
C00604=-22.654,31.927,23.612,177.2881,9.7292,0.0000
C00605=-23.165,33.374,24.311,179.9993,0.0014,0.0000
C00606=-24.090,35.112,25.043,-177.8523,-4.0195,0.0000
C00607=-25.172,37.045,25.615,-176.8232,-6.2765,0.0000
C00608=-26.028,38.969,25.902,-178.5075,-6.9409,0.0000
C00609=-25.888,41.068,26.054,178.6837,-3.9532,0.0000
C00610=-24.719,43.046,26.178,178.5181,-1.6245,0.0000
C00611=-22.710,44.510,26.305,179.8857,-0.0605,0.0000
C00612=-20.355,45.665,26.389,179.9853,-0.0067,0.0000
C00613=-17.897,46.683,26.389,179.9849,-0.0057,0.0000
C00614=-15.415,47.531,26.305,179.8764,-0.0380,0.0000
C00615=-12.959,47.917,26.178,177.8036,0.1012,0.0000
C00616=-10.734,47.345,26.054,176.2738,1.8650,0.0000
C00617=-9.151,45.960,25.902,176.1277,5.9542,0.0000
C00618=-8.395,43.994,25.615,177.7869,6.6761,0.0000
C00619=-7.794,41.862,25.043,178.6707,4.3586,0.0000
C00620=-7.219,39.979,24.311,-179.9995,-0.0014,0.0000
C00621=-6.557,38.594,23.612,-174.9776,-8.7701,0.0000
C00622=-5.504,37.838,23.110,-148.3545,-11.5388,0.0000
C00623=-3.633,37.737,22.912,-141.0650,0.5420,0.0000
C00624=-1.790,37.849,22.904,-140.8005,1.8932,0.0000
C00625=0.000,37.892,22.909,-140.7729,0.0001,0.0000
C00626=0.000,36.499,24.612,-140.7318,-0.0000,0.0000
C00627=1.663,36.461,24.606,-140.7580,-1.8542,0.0000
C00628=3.419,36.362,24.616,-141.0814,-0.0176,0.0000
C00629=5.241,36.506,24.842,-150.1674,13.0548,0.0000
C00630=6.234,37.375,25.413,-176.8918,6.5361,0.0000
C00631=6.845,38.939,26.213,179.5575,-1.4302,0.0000
C00632=7.384,41.061,27.051,178.6140,-5.2236,0.0000
C00633=7.952,43.467,27.704,177.9157,-7.3480,0.0000
C00634=8.667,45.697,28.032,176.2007,-6.7343,0.0000
C00635=10.278,47.290,28.205,175.9685,-2.2766,0.0000
C00636=12.598,47.983,28.348,177.6326,-0.1677,0.0000
C00637=15.186,47.607,28.492,179.8606,0.0424,0.0000
C00638=17.819,46.713,28.587,179.9832,0.0063,0.0000
C00639=20.431,45.631,28.587,179.9837,0.0074,0.0000
C00640=22.925,44.401,28.492,179.8715,0.0686,0.0000
C00641=25.021,42.837,28.348,178.4441,1.7924,0.0000
C00642=26.172,40.707,28.205,178.7594,4.4600,0.0000
C00643=26.184,38.442,28.032,-177.8970,7.4378,0.0000
C00644=25.113,36.359,27.704,-176.2519,6.6580,0.0000
C00645=23.813,34.256,27.051,-177.2773,4.6696,0.0000
C00646=22.694,32.374,26.213,-179.3014,1.3241,0.0000
C00647=22.020,30.836,25.413,177.5527,-6.8102,0.0000
C00648=22.108,29.520,24.842,-167.7845,-30.1586,0.0000
C00649=23.294,28.129,24.616,-150.2640,-26.3593,0.0000
C00650=24.606,26.957,24.606,-148.7370,-25.1000,0.0000
C00651=25.809,25.809,24.612,-149.9675,-26.5875,0.0000
C00652=26.957,24.606,24.606,-151.2768,-28.0317,0.0000
C00653=28.129,23.294,24.616,-150.2872,-26.3854,0.0000
C00654=29.520,22.108,24.842,-149.2681,-10.5421,0.0000
C00655=30.836,22.020,25.413,-173.1836,2.4300,0.0000
C00656=32.374,22.694,26.213,178.6758,-0.6984,0.0000
C00657=34.256,23.813,27.051,175.3251,-2.7137,0.0000
C00658=36.359,25.113,27.704,173.3278,-3.7228,0.0000
C00659=38.442,26.184,28.032,172.5572,-2.0853,0.0000
C00660=40.707,26.172,28.205,175.5389,1.2368,0.0000
C00661=42.837,25.021,28.348,178.2069,1.5552,0.0000
C00662=44.401,22.925,28.492,179.9314,0.1285,0.0000
C00663=45.631,20.431,28.587,179.9926,0.0163,0.0000
C00664=46.713,17.819,28.587,179.9937,0.0168,0.0000
C00665=47.607,15.186,28.492,179.9576,0.1394,0.0000
C00666=47.983,12.598,28.348,-179.8322,2.3674,0.0000
C00667=47.290,10.278,28.205,-177.7177,4.0283,0.0000
C00668=45.697,8.667,28.032,-173.2510,3.7731,0.0000
C00669=43.467,7.952,27.704,-172.6472,2.0672,0.0000
C00670=41.061,7.384,27.051,-174.7748,1.3803,0.0000
C00671=38.939,6.845,26.213,-178.5698,0.4423,0.0000
C00672=37.375,6.234,25.413,173.4543,-3.0880,0.0000
C00673=36.506,5.241,24.842,165.0348,-28.9870,0.0000
C00674=36.362,3.419,24.616,-179.9774,-38.9186,0.0000
C00675=36.461,1.663,24.606,-177.6064,-39.2175,0.0000
C00676=36.499,0.000,24.612,-179.9999,-39.2682,0.0000
C00677=36.461,-1.662,24.606,177.6064,-39.2176,0.0000
C00678=36.362,-3.419,24.616,179.9798,-38.9183,0.0000
C00679=36.506,-5.241,24.842,-165.0352,-28.9875,0.0000
C00680=37.375,-6.234,25.413,-173.4543,-3.0880,0.0000
C00681=38.939,-6.845,26.213,178.5698,0.4423,0.0000
C00682=41.061,-7.384,27.051,174.7748,1.3803,0.0000
C00683=43.467,-7.952,27.704,172.6472,2.0672,0.0000
C00684=45.697,-8.667,28.032,173.2510,3.7731,0.0000
C00685=47.290,-10.278,28.205,177.7177,4.0283,0.0000
C00686=47.983,-12.598,28.348,179.8322,2.3674,0.0000
C00687=47.607,-15.186,28.492,-179.9576,0.1394,0.0000
C00688=46.713,-17.819,28.587,-179.9937,0.0168,0.0000
C00689=45.631,-20.431,28.587,-179.9926,0.0163,0.0000
C00690=44.401,-22.925,28.492,-179.9314,0.1285,0.0000
C00691=42.837,-25.021,28.348,-178.2069,1.5552,0.0000
C00692=40.707,-26.172,28.205,-175.5389,1.2368,0.0000
C00693=38.442,-26.184,28.032,-172.5572,-2.0853,0.0000
C00694=36.359,-25.113,27.704,-173.3278,-3.7228,0.0000
C00695=34.256,-23.813,27.051,-175.3251,-2.7137,0.0000
C00696=32.374,-22.694,26.213,-178.6758,-0.6984,0.0000
C00697=30.836,-22.020,25.413,173.1836,2.4300,0.0000
C00698=29.520,-22.108,24.842,149.2682,-10.5415,0.0000
C00699=28.129,-23.294,24.616,150.2882,-26.3871,0.0000
C00700=26.957,-24.606,24.606,151.2769,-28.0317,0.0000
C00701=25.809,-25.809,24.612,149.9676,-26.5875,0.0000
C00702=24.606,-26.957,24.606,148.7370,-25.1001,0.0000
C00703=23.294,-28.129,24.616,150.2656,-26.3605,0.0000
C00704=22.108,-29.520,24.842,167.7838,-30.1586,0.0000
C00705=22.020,-30.836,25.413,-177.5527,-6.8102,0.0000
C00706=22.694,-32.374,26.213,179.3014,1.3241,0.0000
C00707=23.813,-34.256,27.051,177.2773,4.6696,0.0000
C00708=25.113,-36.359,27.704,176.2519,6.6580,0.0000
C00709=26.184,-38.442,28.032,177.8970,7.4378,0.0000
C00710=26.172,-40.707,28.205,-178.7594,4.4600,0.0000
C00711=25.021,-42.837,28.348,-178.4441,1.7924,0.0000
C00712=22.925,-44.401,28.492,-179.8715,0.0686,0.0000
C00713=20.431,-45.631,28.587,-179.9837,0.0074,0.0000
C00714=17.819,-46.713,28.587,-179.9832,0.0063,0.0000
C00715=15.186,-47.607,28.492,-179.8606,0.0424,0.0000
C00716=12.598,-47.983,28.348,-177.6326,-0.1677,0.0000
C00717=10.278,-47.290,28.205,-175.9685,-2.2766,0.0000
C00718=8.667,-45.697,28.032,-176.2007,-6.7343,0.0000
C00719=7.952,-43.467,27.704,-177.9157,-7.3480,0.0000
C00720=7.384,-41.061,27.051,-178.6140,-5.2236,0.0000
C00721=6.845,-38.939,26.213,-179.5575,-1.4302,0.0000
C00722=6.234,-37.375,25.413,176.8918,6.5361,0.0000
C00723=5.241,-36.506,24.842,150.1674,13.0548,0.0000
C00724=3.419,-36.362,24.616,141.0814,-0.0176,0.0000
C00725=1.663,-36.461,24.606,140.7580,-1.8542,0.0000
C00726=0.000,-36.499,24.612,140.7318,-0.0000,0.0000
C00727=0.000,-36.499,24.612,140.7318,-0.0000,0.0000
C00728=-1.662,-36.461,24.606,140.7579,1.8542,0.0000
C00729=-3.419,-36.362,24.616,141.0817,0.0157,0.0000
C00730=-5.241,-36.506,24.842,150.1669,-13.0544,0.0000
C00731=-6.234,-37.375,25.413,176.8918,-6.5361,0.0000
C00732=-6.845,-38.939,26.213,-179.5575,1.4302,0.0000
C00733=-7.384,-41.061,27.051,-178.6140,5.2236,0.0000
C00734=-7.952,-43.467,27.704,-177.9157,7.3480,0.0000
C00735=-8.667,-45.697,28.032,-176.2007,6.7343,0.0000
C00736=-10.278,-47.290,28.205,-175.9685,2.2766,0.0000
C00737=-12.598,-47.983,28.348,-177.6326,0.1677,0.0000
C00738=-15.186,-47.607,28.492,-179.8606,-0.0424,0.0000
C00739=-17.819,-46.713,28.587,-179.9832,-0.0063,0.0000
C00740=-20.431,-45.631,28.587,-179.9837,-0.0074,0.0000
C00741=-22.925,-44.401,28.492,-179.8715,-0.0686,0.0000
C00742=-25.021,-42.837,28.348,-178.4441,-1.7924,0.0000
C00743=-26.172,-40.707,28.205,-178.7594,-4.4600,0.0000
C00744=-26.184,-38.442,28.032,177.8970,-7.4378,0.0000
C00745=-25.113,-36.359,27.704,176.2519,-6.6580,0.0000
C00746=-23.813,-34.256,27.051,177.2773,-4.6696,0.0000
C00747=-22.694,-32.374,26.213,179.3014,-1.3241,0.0000
C00748=-22.020,-30.836,25.413,-177.5527,6.8102,0.0000
C00749=-22.108,-29.520,24.842,167.7845,30.1586,0.0000
C00750=-23.294,-28.129,24.616,150.2640,26.3593,0.0000
C00751=-24.606,-26.957,24.606,148.7370,25.1000,0.0000
C00752=-25.809,-25.809,24.612,149.9675,26.5875,0.0000
C00753=-26.957,-24.606,24.606,151.2768,28.0317,0.0000
C00754=-28.129,-23.294,24.616,150.2872,26.3854,0.0000
C00755=-29.520,-22.108,24.842,149.2681,10.5421,0.0000
C00756=-30.836,-22.020,25.413,173.1836,-2.4300,0.0000
C00757=-32.374,-22.694,26.213,-178.6758,0.6984,0.0000
C00758=-34.256,-23.813,27.051,-175.3251,2.7137,0.0000
C00759=-36.359,-25.113,27.704,-173.3278,3.7228,0.0000
C00760=-38.442,-26.184,28.032,-172.5572,2.0853,0.0000
C00761=-40.707,-26.172,28.205,-175.5389,-1.2368,0.0000
C00762=-42.837,-25.021,28.348,-178.2069,-1.5552,0.0000
C00763=-44.401,-22.925,28.492,-179.9314,-0.1285,0.0000
C00764=-45.631,-20.431,28.587,-179.9926,-0.0163,0.0000
C00765=-46.713,-17.819,28.587,-179.9937,-0.0168,0.0000
C00766=-47.607,-15.186,28.492,-179.9576,-0.1394,0.0000
C00767=-47.983,-12.598,28.348,179.8322,-2.3674,0.0000
C00768=-47.290,-10.278,28.205,177.7177,-4.0283,0.0000
C00769=-45.697,-8.667,28.032,173.2510,-3.7731,0.0000
C00770=-43.467,-7.952,27.704,172.6472,-2.0672,0.0000
C00771=-41.061,-7.384,27.051,174.7748,-1.3803,0.0000
C00772=-38.939,-6.845,26.213,178.5698,-0.4423,0.0000
C00773=-37.375,-6.234,25.413,-173.4543,3.0880,0.0000
C00774=-36.506,-5.241,24.842,-165.0348,28.9870,0.0000
C00775=-36.362,-3.419,24.616,179.9774,38.9186,0.0000
C00776=-36.461,-1.663,24.606,177.6064,39.2175,0.0000
C00777=-36.499,0.000,24.612,179.9999,39.2682,0.0000
C00778=-36.461,1.662,24.606,-177.6064,39.2176,0.0000
C00779=-36.362,3.419,24.616,-179.9798,38.9183,0.0000
C00780=-36.506,5.241,24.842,165.0352,28.9875,0.0000
C00781=-37.375,6.234,25.413,173.4543,3.0880,0.0000
C00782=-38.939,6.845,26.213,-178.5698,-0.4423,0.0000
C00783=-41.061,7.384,27.051,-174.7748,-1.3803,0.0000
C00784=-43.467,7.952,27.704,-172.6472,-2.0672,0.0000
C00785=-45.697,8.667,28.032,-173.2510,-3.7731,0.0000
C00786=-47.290,10.278,28.205,-177.7177,-4.0283,0.0000
C00787=-47.983,12.598,28.348,-179.8322,-2.3674,0.0000
C00788=-47.607,15.186,28.492,179.9576,-0.1394,0.0000
C00789=-46.713,17.819,28.587,179.9937,-0.0168,0.0000
C00790=-45.631,20.431,28.587,179.9926,-0.0163,0.0000
C00791=-44.401,22.925,28.492,179.9314,-0.1285,0.0000
C00792=-42.837,25.021,28.348,178.2069,-1.5552,0.0000
C00793=-40.707,26.172,28.205,175.5389,-1.2368,0.0000
C00794=-38.442,26.184,28.032,172.5572,2.0853,0.0000
C00795=-36.359,25.113,27.704,173.3278,3.7228,0.0000
C00796=-34.256,23.813,27.051,175.3251,2.7137,0.0000
C00797=-32.374,22.694,26.213,178.6758,0.6984,0.0000
C00798=-30.836,22.020,25.413,-173.1836,-2.4300,0.0000
C00799=-29.520,22.108,24.842,-149.2682,10.5415,0.0000
C00800=-28.129,23.294,24.616,-150.2882,26.3871,0.0000
C00801=-26.957,24.606,24.606,-151.2769,28.0317,0.0000
C00802=-25.809,25.809,24.612,-149.9676,26.5875,0.0000
C00803=-24.606,26.957,24.606,-148.7370,25.1001,0.0000
C00804=-23.294,28.129,24.616,-150.2656,26.3605,0.0000
C00805=-22.108,29.520,24.842,-167.7838,30.1586,0.0000
C00806=-22.020,30.836,25.413,177.5527,6.8102,0.0000
C00807=-22.694,32.374,26.213,-179.3014,-1.3241,0.0000
C00808=-23.813,34.256,27.051,-177.2773,-4.6696,0.0000
C00809=-25.113,36.359,27.704,-176.2519,-6.6580,0.0000
C00810=-26.184,38.442,28.032,-177.8970,-7.4378,0.0000
C00811=-26.172,40.707,28.205,178.7594,-4.4600,0.0000
C00812=-25.021,42.837,28.348,178.4441,-1.7924,0.0000
C00813=-22.925,44.401,28.492,179.8715,-0.0686,0.0000
C00814=-20.431,45.631,28.587,179.9837,-0.0074,0.0000
C00815=-17.819,46.713,28.587,179.9832,-0.0063,0.0000
C00816=-15.186,47.607,28.492,179.8606,-0.0424,0.0000
C00817=-12.598,47.983,28.348,177.6326,0.1677,0.0000
C00818=-10.278,47.290,28.205,175.9685,2.2766,0.0000
C00819=-8.667,45.697,28.032,176.2007,6.7343,0.0000
C00820=-7.952,43.467,27.704,177.9157,7.3480,0.0000
C00821=-7.384,41.061,27.051,178.6140,5.2236,0.0000
C00822=-6.845,38.939,26.213,179.5575,1.4302,0.0000
C00823=-6.234,37.375,25.413,-176.8918,-6.5361,0.0000
C00824=-5.241,36.506,24.842,-150.1669,-13.0544,0.0000
C00825=-3.419,36.362,24.616,-141.0817,0.0157,0.0000
C00826=-1.662,36.461,24.606,-140.7579,1.8542,0.0000
C00827=0.000,36.499,24.612,-140.7318,-0.0000,0.0000
C00828=0.000,35.110,26.318,-140.9850,-0.0002,0.0000
C00829=1.536,35.076,26.311,-141.0094,-1.7975,0.0000
C00830=3.206,34.989,26.322,-141.4086,0.5388,0.0000
C00831=4.979,35.179,26.576,-152.4042,14.1984,0.0000
C00832=5.912,36.162,27.221,-178.2378,4.4014,0.0000
C00833=6.475,37.910,28.122,179.3106,-2.5546,0.0000
C00834=6.981,40.274,29.065,178.6436,-5.7923,0.0000
C00835=7.520,42.952,29.799,178.1039,-7.6946,0.0000
C00836=8.198,45.442,30.166,176.4208,-7.1814,0.0000
C00837=9.836,47.237,30.360,175.8447,-2.5886,0.0000
C00838=12.248,48.046,30.519,177.5461,-0.2273,0.0000
C00839=14.965,47.679,30.679,179.8510,0.0449,0.0000
C00840=17.744,46.742,30.786,179.9823,0.0066,0.0000
C00841=20.505,45.599,30.786,179.9828,0.0078,0.0000
C00842=23.132,44.297,30.679,179.8629,0.0736,0.0000
C00843=25.313,42.634,30.519,178.4250,1.8958,0.0000
C00844=26.446,40.357,30.360,178.8932,4.7680,0.0000
C00845=26.335,37.929,30.166,-177.4211,7.5964,0.0000
C00846=25.054,35.689,29.799,-175.8715,6.7687,0.0000
C00847=23.542,33.414,29.065,-176.8516,5.0495,0.0000
C00848=22.228,31.385,28.122,-178.6801,2.2934,0.0000
C00849=21.390,29.751,27.221,178.1272,-4.3556,0.0000
C00850=21.354,28.396,26.576,-170.4783,-29.4055,0.0000
C00851=22.474,27.008,26.322,-150.9350,-26.5960,0.0000
C00852=23.717,25.889,26.311,-148.9957,-24.9930,0.0000
C00853=24.826,24.826,26.318,-150.1910,-26.4322,0.0000
C00854=25.888,23.717,26.311,-151.4600,-27.8313,0.0000
C00855=27.008,22.474,26.322,-150.1945,-25.7451,0.0000
C00856=28.396,21.354,26.576,-150.2532,-8.2862,0.0000
C00857=29.751,21.390,27.221,-175.6421,1.8674,0.0000
C00858=31.385,22.228,28.122,177.7060,-1.3189,0.0000
C00859=33.414,23.542,29.065,174.9429,-3.1362,0.0000
C00860=35.689,25.054,29.799,173.2138,-4.0997,0.0000
C00861=37.929,26.335,30.166,172.3960,-2.5562,0.0000
C00862=40.357,26.446,30.360,175.2311,1.1029,0.0000
C00863=42.634,25.313,30.519,178.1035,1.5741,0.0000
C00864=44.297,23.132,30.679,179.9264,0.1371,0.0000
C00865=45.599,20.505,30.786,179.9922,0.0172,0.0000
C00866=46.742,17.744,30.786,179.9934,0.0177,0.0000
C00867=47.679,14.965,30.679,179.9551,0.1490,0.0000
C00868=48.046,12.248,30.519,-179.7724,2.4539,0.0000
C00869=47.237,9.836,30.360,-177.4046,4.1511,0.0000
C00870=45.442,8.198,30.166,-172.8047,3.5511,0.0000
C00871=42.952,7.520,29.799,-172.3012,1.8790,0.0000
C00872=40.274,6.981,29.065,-174.2061,1.3495,0.0000
C00873=37.910,6.475,28.122,-177.4452,0.6888,0.0000
C00874=36.162,5.912,27.221,175.5965,-1.7570,0.0000
C00875=35.179,4.979,26.576,164.0667,-26.6847,0.0000
C00876=34.989,3.206,26.322,179.3106,-38.5893,0.0000
C00877=35.076,1.536,26.311,-177.6879,-38.9678,0.0000
C00878=35.110,0.000,26.318,-179.9997,-39.0150,0.0000
C00879=35.076,-1.535,26.311,177.6876,-38.9678,0.0000
C00880=34.989,-3.206,26.322,-179.3080,-38.5889,0.0000
C00881=35.179,-4.979,26.576,-164.0669,-26.6851,0.0000
C00882=36.162,-5.912,27.221,-175.5965,-1.7570,0.0000
C00883=37.910,-6.475,28.122,177.4452,0.6888,0.0000
C00884=40.274,-6.981,29.065,174.2061,1.3495,0.0000
C00885=42.952,-7.520,29.799,172.3012,1.8790,0.0000
C00886=45.442,-8.198,30.166,172.8047,3.5511,0.0000
C00887=47.237,-9.836,30.360,177.4046,4.1511,0.0000
C00888=48.046,-12.248,30.519,179.7724,2.4539,0.0000
C00889=47.679,-14.965,30.679,-179.9551,0.1490,0.0000
C00890=46.742,-17.744,30.786,-179.9934,0.0177,0.0000
C00891=45.599,-20.505,30.786,-179.9922,0.0172,0.0000
C00892=44.297,-23.132,30.679,-179.9264,0.1371,0.0000
C00893=42.634,-25.313,30.519,-178.1035,1.5741,0.0000
C00894=40.357,-26.446,30.360,-175.2311,1.1029,0.0000
C00895=37.929,-26.335,30.166,-172.3960,-2.5562,0.0000
C00896=35.689,-25.054,29.799,-173.2138,-4.0997,0.0000
C00897=33.414,-23.542,29.065,-174.9429,-3.1362,0.0000
C00898=31.385,-22.228,28.122,-177.7060,-1.3189,0.0000
C00899=29.751,-21.390,27.221,175.6421,1.8674,0.0000
C00900=28.396,-21.354,26.576,150.2533,-8.2857,0.0000
C00901=27.008,-22.474,26.322,150.1955,-25.7469,0.0000
C00902=25.889,-23.717,26.311,151.4600,-27.8311,0.0000
C00903=24.826,-24.826,26.318,150.1913,-26.4325,0.0000
C00904=23.717,-25.888,26.311,148.9956,-24.9929,0.0000
C00905=22.474,-27.008,26.322,150.9367,-26.5973,0.0000
C00906=21.354,-28.396,26.576,170.4778,-29.4056,0.0000
C00907=21.390,-29.751,27.221,-178.1272,-4.3556,0.0000
C00908=22.228,-31.385,28.122,178.6801,2.2934,0.0000
C00909=23.542,-33.414,29.065,176.8516,5.0495,0.0000
C00910=25.054,-35.689,29.799,175.8715,6.7687,0.0000
C00911=26.335,-37.929,30.166,177.4211,7.5964,0.0000
C00912=26.446,-40.357,30.360,-178.8932,4.7680,0.0000
C00913=25.313,-42.634,30.519,-178.4250,1.8958,0.0000
C00914=23.132,-44.297,30.679,-179.8629,0.0736,0.0000
C00915=20.505,-45.599,30.786,-179.9828,0.0078,0.0000
C00916=17.744,-46.742,30.786,-179.9823,0.0066,0.0000
C00917=14.965,-47.679,30.679,-179.8510,0.0449,0.0000
C00918=12.248,-48.046,30.519,-177.5461,-0.2273,0.0000
C00919=9.836,-47.237,30.360,-175.8447,-2.5886,0.0000
C00920=8.198,-45.442,30.166,-176.4208,-7.1814,0.0000
C00921=7.520,-42.952,29.799,-178.1039,-7.6946,0.0000
C00922=6.981,-40.274,29.065,-178.6436,-5.7923,0.0000
C00923=6.475,-37.910,28.122,-179.3106,-2.5546,0.0000
C00924=5.912,-36.162,27.221,178.2378,4.4014,0.0000
C00925=4.979,-35.179,26.576,152.4042,14.1984,0.0000
C00926=3.206,-34.989,26.322,141.4086,0.5388,0.0000
C00927=1.536,-35.076,26.311,141.0094,-1.7975,0.0000
C00928=0.000,-35.110,26.318,140.9850,-0.0002,0.0000
C00929=0.000,-35.110,26.318,140.9850,-0.0002,0.0000
C00930=-1.535,-35.076,26.311,141.0094,1.7977,0.0000
C00931=-3.206,-34.989,26.322,141.4090,-0.5409,0.0000
C00932=-4.979,-35.179,26.576,152.4038,-14.1981,0.0000
C00933=-5.912,-36.162,27.221,178.2378,-4.4014,0.0000
C00934=-6.475,-37.910,28.122,-179.3106,2.5546,0.0000
C00935=-6.981,-40.274,29.065,-178.6436,5.7923,0.0000
C00936=-7.520,-42.952,29.799,-178.1039,7.6946,0.0000
C00937=-8.198,-45.442,30.166,-176.4208,7.1814,0.0000
C00938=-9.836,-47.237,30.360,-175.8447,2.5886,0.0000
C00939=-12.248,-48.046,30.519,-177.5461,0.2273,0.0000
C00940=-14.965,-47.679,30.679,-179.8510,-0.0449,0.0000
C00941=-17.744,-46.742,30.786,-179.9823,-0.0066,0.0000
C00942=-20.505,-45.599,30.786,-179.9828,-0.0078,0.0000
C00943=-23.132,-44.297,30.679,-179.8629,-0.0736,0.0000
C00944=-25.313,-42.634,30.519,-178.4250,-1.8958,0.0000
C00945=-26.446,-40.357,30.360,-178.8932,-4.7680,0.0000
C00946=-26.335,-37.929,30.166,177.4211,-7.5964,0.0000
C00947=-25.054,-35.689,29.799,175.8715,-6.7687,0.0000
C00948=-23.542,-33.414,29.065,176.8516,-5.0495,0.0000
C00949=-22.228,-31.385,28.122,178.6801,-2.2934,0.0000
C00950=-21.390,-29.751,27.221,-178.1272,4.3556,0.0000
C00951=-21.354,-28.396,26.576,170.4783,29.4055,0.0000
C00952=-22.474,-27.008,26.322,150.9350,26.5960,0.0000
C00953=-23.717,-25.889,26.311,148.9957,24.9930,0.0000
C00954=-24.826,-24.826,26.318,150.1910,26.4322,0.0000
C00955=-25.888,-23.717,26.311,151.4600,27.8313,0.0000
C00956=-27.008,-22.474,26.322,150.1945,25.7451,0.0000
C00957=-28.396,-21.354,26.576,150.2532,8.2862,0.0000
C00958=-29.751,-21.390,27.221,175.6421,-1.8674,0.0000
C00959=-31.385,-22.228,28.122,-177.7060,1.3189,0.0000
C00960=-33.414,-23.542,29.065,-174.9429,3.1362,0.0000
C00961=-35.689,-25.054,29.799,-173.2138,4.0997,0.0000
C00962=-37.929,-26.335,30.166,-172.3960,2.5562,0.0000
C00963=-40.357,-26.446,30.360,-175.2311,-1.1029,0.0000
C00964=-42.634,-25.313,30.519,-178.1035,-1.5741,0.0000
C00965=-44.297,-23.132,30.679,-179.9264,-0.1371,0.0000
C00966=-45.599,-20.505,30.786,-179.9922,-0.0172,0.0000
C00967=-46.742,-17.744,30.786,-179.9934,-0.0177,0.0000
C00968=-47.679,-14.965,30.679,-179.9551,-0.1490,0.0000
C00969=-48.046,-12.248,30.519,179.7724,-2.4539,0.0000
C00970=-47.237,-9.836,30.360,177.4046,-4.1511,0.0000
C00971=-45.442,-8.198,30.166,172.8047,-3.5511,0.0000
C00972=-42.952,-7.520,29.799,172.3012,-1.8790,0.0000
C00973=-40.274,-6.981,29.065,174.2061,-1.3495,0.0000
C00974=-37.910,-6.475,28.122,177.4452,-0.6888,0.0000
C00975=-36.162,-5.912,27.221,-175.5965,1.7570,0.0000
C00976=-35.179,-4.979,26.576,-164.0667,26.6847,0.0000
C00977=-34.989,-3.206,26.322,-179.3106,38.5893,0.0000
C00978=-35.076,-1.536,26.311,177.6879,38.9678,0.0000
C00979=-35.110,0.000,26.318,179.9997,39.0150,0.0000
C00980=-35.076,1.535,26.311,-177.6876,38.9678,0.0000
C00981=-34.989,3.206,26.322,179.3080,38.5889,0.0000
C00982=-35.179,4.979,26.576,164.0669,26.6851,0.0000
C00983=-36.162,5.912,27.221,175.5965,1.7570,0.0000
C00984=-37.910,6.475,28.122,-177.4452,-0.6888,0.0000
C00985=-40.274,6.981,29.065,-174.2061,-1.3495,0.0000
C00986=-42.952,7.520,29.799,-172.3012,-1.8790,0.0000
C00987=-45.442,8.198,30.166,-172.8047,-3.5511,0.0000
C00988=-47.237,9.836,30.360,-177.4046,-4.1511,0.0000
C00989=-48.046,12.248,30.519,-179.7724,-2.4539,0.0000
C00990=-47.679,14.965,30.679,179.9551,-0.1490,0.0000
C00991=-46.742,17.744,30.786,179.9934,-0.0177,0.0000
C00992=-45.599,20.505,30.786,179.9922,-0.0172,0.0000
C00993=-44.297,23.132,30.679,179.9264,-0.1371,0.0000
C00994=-42.634,25.313,30.519,178.1035,-1.5741,0.0000
C00995=-40.357,26.446,30.360,175.2311,-1.1029,0.0000
C00996=-37.929,26.335,30.166,172.3960,2.5562,0.0000
C00997=-35.689,25.054,29.799,173.2138,4.0997,0.0000
C00998=-33.414,23.542,29.065,174.9429,3.1362,0.0000
C00999=-31.385,22.228,28.122,177.7060,1.3189,0.0000
C01000=-29.751,21.390,27.221,-175.6421,-1.8674,0.0000
C01001=-28.396,21.354,26.576,-150.2533,8.2857,0.0000
C01002=-27.008,22.474,26.322,-150.1955,25.7469,0.0000
C01003=-25.889,23.717,26.311,-151.4600,27.8311,0.0000
C01004=-24.826,24.826,26.318,-150.1913,26.4325,0.0000
C01005=-23.717,25.888,26.311,-148.9956,24.9929,0.0000
C01006=-22.474,27.008,26.322,-150.9367,26.5973,0.0000
C01007=-21.354,28.396,26.576,-170.4778,29.4056,0.0000
C01008=-21.390,29.751,27.221,178.1272,4.3556,0.0000
C01009=-22.228,31.385,28.122,-178.6801,-2.2934,0.0000
C01010=-23.542,33.414,29.065,-176.8516,-5.0495,0.0000
C01011=-25.054,35.689,29.799,-175.8715,-6.7687,0.0000
C01012=-26.335,37.929,30.166,-177.4211,-7.5964,0.0000
C01013=-26.446,40.357,30.360,178.8932,-4.7680,0.0000
C01014=-25.313,42.634,30.519,178.4250,-1.8958,0.0000
C01015=-23.132,44.297,30.679,179.8629,-0.0736,0.0000
C01016=-20.505,45.599,30.786,179.9828,-0.0078,0.0000
C01017=-17.744,46.742,30.786,179.9823,-0.0066,0.0000
C01018=-14.965,47.679,30.679,179.8510,-0.0449,0.0000
C01019=-12.248,48.046,30.519,177.5461,0.2273,0.0000
C01020=-9.836,47.237,30.360,175.8447,2.5886,0.0000
C01021=-8.198,45.442,30.166,176.4208,7.1814,0.0000
C01022=-7.520,42.952,29.799,178.1039,7.6946,0.0000
C01023=-6.981,40.274,29.065,178.6436,5.7923,0.0000
C01024=-6.475,37.910,28.122,179.3106,2.5546,0.0000
C01025=-5.912,36.162,27.221,-178.2378,-4.4014,0.0000
C01026=-4.979,35.179,26.576,-152.4038,-14.1981,0.0000
C01027=-3.206,34.989,26.322,-141.4090,-0.5409,0.0000
C01028=-1.535,35.076,26.311,-141.0094,1.7977,0.0000
C01029=0.000,35.110,26.318,-140.9850,-0.0002,0.0000
C01030=0.000,33.732,28.034,-141.5426,-0.0004,0.0000
C01031=1.410,33.704,28.025,-141.5650,-1.7225,0.0000
C01032=2.994,33.629,28.038,-142.0582,1.1123,0.0000
C01033=4.720,33.865,28.321,-154.9684,14.9015,0.0000
C01034=5.595,34.967,29.040,-179.1465,2.5036,0.0000
C01035=6.113,36.903,30.045,179.1942,-3.3819,0.0000
C01036=6.591,39.512,31.092,178.7262,-6.0852,0.0000
C01037=7.106,42.459,31.903,178.3205,-7.7402,0.0000
C01038=7.750,45.198,32.306,176.7329,-7.3046,0.0000
C01039=9.416,47.186,32.519,175.8897,-2.7751,0.0000
C01040=11.916,48.107,32.693,177.5484,-0.2738,0.0000
C01041=14.756,47.748,32.868,179.8479,0.0454,0.0000
C01042=17.673,46.769,32.984,179.9821,0.0067,0.0000
C01043=20.574,45.568,32.984,179.9826,0.0079,0.0000
C01044=23.329,44.198,32.868,179.8603,0.0754,0.0000
C01045=25.591,42.442,32.693,178.4595,1.9270,0.0000
C01046=26.708,40.024,32.519,179.0576,4.8679,0.0000
C01047=26.480,37.440,32.306,-177.1134,7.4624,0.0000
C01048=24.998,35.047,31.903,-175.6871,6.6481,0.0000
C01049=23.279,32.600,31.092,-176.5847,5.1975,0.0000
C01050=21.772,30.417,30.045,-178.1760,2.9601,0.0000
C01051=20.769,28.682,29.040,178.8321,-2.3734,0.0000
C01052=20.608,27.283,28.321,-173.0142,-28.0970,0.0000
C01053=21.662,25.896,28.038,-151.9028,-26.6422,0.0000
C01054=22.835,24.829,28.025,-149.5319,-24.7149,0.0000
C01055=23.852,23.852,28.034,-150.6812,-26.0891,0.0000
C01056=24.829,22.835,28.025,-151.8978,-27.4269,0.0000
C01057=25.896,21.662,28.038,-150.3718,-24.8935,0.0000
C01058=27.283,20.608,28.321,-151.7252,-6.1593,0.0000
C01059=28.682,20.769,29.040,-177.6261,1.1669,0.0000
C01060=30.417,21.772,30.045,177.0384,-1.8215,0.0000
C01061=32.600,23.279,31.092,174.7934,-3.4012,0.0000
C01062=35.047,24.998,31.903,173.3332,-4.2839,0.0000
C01063=37.440,26.480,32.306,172.5282,-2.8621,0.0000
C01064=40.024,26.708,32.519,175.1314,0.9390,0.0000
C01065=42.442,25.591,32.693,178.0724,1.5396,0.0000
C01066=44.198,23.329,32.868,179.9246,0.1397,0.0000
C01067=45.568,20.574,32.984,179.9921,0.0174,0.0000
C01068=46.769,17.673,32.984,179.9933,0.0179,0.0000
C01069=47.748,14.756,32.868,179.9546,0.1521,0.0000
C01070=48.107,11.916,32.693,-179.7260,2.4516,0.0000
C01071=47.186,9.416,32.519,-177.2177,4.1055,0.0000
C01072=45.198,7.750,32.306,-172.6836,3.2406,0.0000
C01073=42.459,7.106,31.903,-172.2565,1.6642,0.0000
C01074=39.512,6.591,31.092,-173.9134,1.2666,0.0000
C01075=36.903,6.113,30.045,-176.6177,0.8044,0.0000
C01076=34.967,5.595,29.040,177.4961,-0.8527,0.0000
C01077=33.865,4.720,28.321,163.6329,-24.1350,0.0000
C01078=33.629,2.994,28.038,178.5897,-37.9334,0.0000
C01079=33.704,1.410,28.025,-177.8015,-38.4145,0.0000
C01080=33.732,0.000,28.034,-179.9996,-38.4574,0.0000
C01081=33.704,-1.410,28.025,177.8010,-38.4145,0.0000
C01082=33.629,-2.994,28.038,-178.5870,-37.9329,0.0000
C01083=33.865,-4.720,28.321,-163.6330,-24.1352,0.0000
C01084=34.967,-5.595,29.040,-177.4961,-0.8527,0.0000
C01085=36.903,-6.113,30.045,176.6177,0.8044,0.0000
C01086=39.512,-6.591,31.092,173.9134,1.2666,0.0000
C01087=42.459,-7.106,31.903,172.2565,1.6642,0.0000
C01088=45.198,-7.750,32.306,172.6836,3.2406,0.0000
C01089=47.186,-9.416,32.519,177.2177,4.1055,0.0000
C01090=48.107,-11.916,32.693,179.7260,2.4516,0.0000
C01091=47.748,-14.756,32.868,-179.9546,0.1521,0.0000
C01092=46.769,-17.673,32.984,-179.9933,0.0179,0.0000
C01093=45.568,-20.574,32.984,-179.9921,0.0174,0.0000
C01094=44.198,-23.329,32.868,-179.9246,0.1397,0.0000
C01095=42.442,-25.591,32.693,-178.0724,1.5396,0.0000
C01096=40.024,-26.708,32.519,-175.1314,0.9390,0.0000
C01097=37.440,-26.480,32.306,-172.5282,-2.8621,0.0000
C01098=35.047,-24.998,31.903,-173.3332,-4.2839,0.0000
C01099=32.600,-23.279,31.092,-174.7934,-3.4012,0.0000
C01100=30.417,-21.772,30.045,-177.0384,-1.8215,0.0000
C01101=28.682,-20.769,29.040,177.6261,1.1669,0.0000
C01102=27.283,-20.608,28.321,151.7253,-6.1591,0.0000
C01103=25.896,-21.662,28.038,150.3728,-24.8955,0.0000
C01104=24.829,-22.835,28.025,151.8976,-27.4266,0.0000
C01105=23.852,-23.852,28.034,150.6816,-26.0897,0.0000
C01106=22.835,-24.829,28.025,149.5316,-24.7147,0.0000
C01107=21.662,-25.896,28.038,151.9047,-26.6435,0.0000
C01108=20.608,-27.283,28.321,173.0140,-28.0971,0.0000
C01109=20.769,-28.682,29.040,-178.8321,-2.3734,0.0000
C01110=21.772,-30.417,30.045,178.1760,2.9601,0.0000
C01111=23.279,-32.600,31.092,176.5847,5.1975,0.0000
C01112=24.998,-35.047,31.903,175.6871,6.6481,0.0000
C01113=26.480,-37.440,32.306,177.1134,7.4624,0.0000
C01114=26.708,-40.024,32.519,-179.0576,4.8679,0.0000
C01115=25.591,-42.442,32.693,-178.4595,1.9270,0.0000
C01116=23.329,-44.198,32.868,-179.8603,0.0754,0.0000
C01117=20.574,-45.568,32.984,-179.9826,0.0079,0.0000
C01118=17.673,-46.769,32.984,-179.9821,0.0067,0.0000
C01119=14.756,-47.748,32.868,-179.8479,0.0454,0.0000
C01120=11.916,-48.107,32.693,-177.5484,-0.2738,0.0000
C01121=9.416,-47.186,32.519,-175.8897,-2.7751,0.0000
C01122=7.750,-45.198,32.306,-176.7329,-7.3046,0.0000
C01123=7.106,-42.459,31.903,-178.3205,-7.7402,0.0000
C01124=6.591,-39.512,31.092,-178.7262,-6.0852,0.0000
C01125=6.113,-36.903,30.045,-179.1942,-3.3819,0.0000
C01126=5.595,-34.967,29.040,179.1465,2.5036,0.0000
C01127=4.720,-33.865,28.321,154.9684,14.9015,0.0000
C01128=2.994,-33.629,28.038,142.0582,1.1123,0.0000
C01129=1.410,-33.704,28.025,141.5650,-1.7225,0.0000
C01130=0.000,-33.732,28.034,141.5426,-0.0004,0.0000
C01131=0.000,-33.732,28.034,141.5426,-0.0004,0.0000
C01132=-1.410,-33.704,28.025,141.5649,1.7228,0.0000
C01133=-2.994,-33.629,28.038,142.0586,-1.1144,0.0000
C01134=-4.720,-33.865,28.321,154.9682,-14.9013,0.0000
C01135=-5.595,-34.967,29.040,179.1465,-2.5036,0.0000
C01136=-6.113,-36.903,30.045,-179.1942,3.3819,0.0000
C01137=-6.591,-39.512,31.092,-178.7262,6.0852,0.0000
C01138=-7.106,-42.459,31.903,-178.3205,7.7402,0.0000
C01139=-7.750,-45.198,32.306,-176.7329,7.3046,0.0000
C01140=-9.416,-47.186,32.519,-175.8897,2.7751,0.0000
C01141=-11.916,-48.107,32.693,-177.5484,0.2738,0.0000
C01142=-14.756,-47.748,32.868,-179.8479,-0.0454,0.0000
C01143=-17.673,-46.769,32.984,-179.9821,-0.0067,0.0000
C01144=-20.574,-45.568,32.984,-179.9826,-0.0079,0.0000
C01145=-23.329,-44.198,32.868,-179.8603,-0.0754,0.0000
C01146=-25.591,-42.442,32.693,-178.4595,-1.9270,0.0000
C01147=-26.708,-40.024,32.519,-179.0576,-4.8679,0.0000
C01148=-26.480,-37.440,32.306,177.1134,-7.4624,0.0000
C01149=-24.998,-35.047,31.903,175.6871,-6.6481,0.0000
C01150=-23.279,-32.600,31.092,176.5847,-5.1975,0.0000
C01151=-21.772,-30.417,30.045,178.1760,-2.9601,0.0000
C01152=-20.769,-28.682,29.040,-178.8321,2.3734,0.0000
C01153=-20.608,-27.283,28.321,173.0142,28.0970,0.0000
C01154=-21.662,-25.896,28.038,151.9028,26.6422,0.0000
C01155=-22.835,-24.829,28.025,149.5319,24.7149,0.0000
C01156=-23.852,-23.852,28.034,150.6812,26.0891,0.0000
C01157=-24.829,-22.835,28.025,151.8978,27.4269,0.0000
C01158=-25.896,-21.662,28.038,150.3718,24.8935,0.0000
C01159=-27.283,-20.608,28.321,151.7252,6.1593,0.0000
C01160=-28.682,-20.769,29.040,177.6261,-1.1669,0.0000
C01161=-30.417,-21.772,30.045,-177.0384,1.8215,0.0000
C01162=-32.600,-23.279,31.092,-174.7934,3.4012,0.0000
C01163=-35.047,-24.998,31.903,-173.3332,4.2839,0.0000
C01164=-37.440,-26.480,32.306,-172.5282,2.8621,0.0000
C01165=-40.024,-26.708,32.519,-175.1314,-0.9390,0.0000
C01166=-42.442,-25.591,32.693,-178.0724,-1.5396,0.0000
C01167=-44.198,-23.329,32.868,-179.9246,-0.1397,0.0000
C01168=-45.568,-20.574,32.984,-179.9921,-0.0174,0.0000
C01169=-46.769,-17.673,32.984,-179.9933,-0.0179,0.0000
C01170=-47.748,-14.756,32.868,-179.9546,-0.1521,0.0000
C01171=-48.107,-11.916,32.693,179.7260,-2.4516,0.0000
C01172=-47.186,-9.416,32.519,177.2177,-4.1055,0.0000
C01173=-45.198,-7.750,32.306,172.6836,-3.2406,0.0000
C01174=-42.459,-7.106,31.903,172.2565,-1.6642,0.0000
C01175=-39.512,-6.591,31.092,173.9134,-1.2666,0.0000
C01176=-36.903,-6.113,30.045,176.6177,-0.8044,0.0000
C01177=-34.967,-5.595,29.040,-177.4961,0.8527,0.0000
C01178=-33.865,-4.720,28.321,-163.6329,24.1350,0.0000
C01179=-33.629,-2.994,28.038,-178.5897,37.9334,0.0000
C01180=-33.704,-1.410,28.025,177.8015,38.4145,0.0000
C01181=-33.732,0.000,28.034,179.9996,38.4574,0.0000
C01182=-33.704,1.410,28.025,-177.8010,38.4145,0.0000
C01183=-33.629,2.994,28.038,178.5870,37.9329,0.0000
C01184=-33.865,4.720,28.321,163.6330,24.1352,0.0000
C01185=-34.967,5.595,29.040,177.4961,0.8527,0.0000
C01186=-36.903,6.113,30.045,-176.6177,-0.8044,0.0000
C01187=-39.512,6.591,31.092,-173.9134,-1.2666,0.0000
C01188=-42.459,7.106,31.903,-172.2565,-1.6642,0.0000
C01189=-45.198,7.750,32.306,-172.6836,-3.2406,0.0000
C01190=-47.186,9.416,32.519,-177.2177,-4.1055,0.0000
C01191=-48.107,11.916,32.693,-179.7260,-2.4516,0.0000
C01192=-47.748,14.756,32.868,179.9546,-0.1521,0.0000
C01193=-46.769,17.673,32.984,179.9933,-0.0179,0.0000
C01194=-45.568,20.574,32.984,179.9921,-0.0174,0.0000
C01195=-44.198,23.329,32.868,179.9246,-0.1397,0.0000
C01196=-42.442,25.591,32.693,178.0724,-1.5396,0.0000
C01197=-40.024,26.708,32.519,175.1314,-0.9390,0.0000
C01198=-37.440,26.480,32.306,172.5282,2.8621,0.0000
C01199=-35.047,24.998,31.903,173.3332,4.2839,0.0000
C01200=-32.600,23.279,31.092,174.7934,3.4012,0.0000
C01201=-30.417,21.772,30.045,177.0384,1.8215,0.0000
C01202=-28.682,20.769,29.040,-177.6261,-1.1669,0.0000
C01203=-27.283,20.608,28.321,-151.7253,6.1591,0.0000
C01204=-25.896,21.662,28.038,-150.3728,24.8955,0.0000
C01205=-24.829,22.835,28.025,-151.8976,27.4266,0.0000
C01206=-23.852,23.852,28.034,-150.6816,26.0897,0.0000
C01207=-22.835,24.829,28.025,-149.5316,24.7147,0.0000
C01208=-21.662,25.896,28.038,-151.9047,26.6435,0.0000
C01209=-20.608,27.283,28.321,-173.0140,28.0971,0.0000
C01210=-20.769,28.682,29.040,178.8321,2.3734,0.0000
C01211=-21.772,30.417,30.045,-178.1760,-2.9601,0.0000
C01212=-23.279,32.600,31.092,-176.5847,-5.1975,0.0000
C01213=-24.998,35.047,31.903,-175.6871,-6.6481,0.0000
C01214=-26.480,37.440,32.306,-177.1134,-7.4624,0.0000
C01215=-26.708,40.024,32.519,179.0576,-4.8679,0.0000
C01216=-25.591,42.442,32.693,178.4595,-1.9270,0.0000
C01217=-23.329,44.198,32.868,179.8603,-0.0754,0.0000
C01218=-20.574,45.568,32.984,179.9826,-0.0079,0.0000
C01219=-17.673,46.769,32.984,179.9821,-0.0067,0.0000
C01220=-14.756,47.748,32.868,179.8479,-0.0454,0.0000
C01221=-11.916,48.107,32.693,177.5484,0.2738,0.0000
C01222=-9.416,47.186,32.519,175.8897,2.7751,0.0000
C01223=-7.750,45.198,32.306,176.7329,7.3046,0.0000
C01224=-7.106,42.459,31.903,178.3205,7.7402,0.0000
C01225=-6.591,39.512,31.092,178.7262,6.0852,0.0000
C01226=-6.113,36.903,30.045,179.1942,3.3819,0.0000
C01227=-5.595,34.967,29.040,-179.1465,-2.5036,0.0000
C01228=-4.720,33.865,28.321,-154.9682,-14.9013,0.0000
C01229=-2.994,33.629,28.038,-142.0586,-1.1144,0.0000
C01230=-1.410,33.704,28.025,-141.5649,1.7228,0.0000
C01231=0.000,33.732,28.034,-141.5426,-0.0004,0.0000
C01232=0.000,32.376,29.766,-142.4274,-0.0005,0.0000
C01233=1.286,32.352,29.757,-142.4475,-1.6281,0.0000
C01234=2.786,32.290,29.771,-143.0534,1.6857,0.0000
C01235=4.465,32.574,30.085,-157.7490,15.1242,0.0000
C01236=5.286,33.800,30.880,-179.7331,0.9107,0.0000
C01237=5.763,35.931,31.987,179.1649,-3.9270,0.0000
C01238=6.219,38.785,33.135,178.8416,-6.1191,0.0000
C01239=6.715,41.994,34.017,178.5475,-7.5040,0.0000
C01240=7.331,44.970,34.453,177.1015,-7.1192,0.0000
C01241=9.024,47.139,34.683,176.0894,-2.8205,0.0000
C01242=11.608,48.163,34.870,177.6414,-0.3019,0.0000
C01243=14.563,47.812,35.059,179.8514,0.0441,0.0000
C01244=17.608,46.795,35.183,179.9827,0.0065,0.0000
C01245=20.638,45.540,35.183,179.9832,0.0077,0.0000
C01246=23.511,44.106,35.059,179.8638,0.0739,0.0000
C01247=25.848,42.264,34.870,178.5453,1.8811,0.0000
C01248=26.951,39.714,34.683,179.2311,4.7588,0.0000
C01249=26.615,36.982,34.453,-176.9875,7.0718,0.0000
C01250=24.946,34.442,34.017,-175.6970,6.3219,0.0000
C01251=23.028,31.823,33.135,-176.4794,5.1399,0.0000
C01252=21.332,29.482,31.987,-177.8101,3.3656,0.0000
C01253=20.163,27.638,30.880,179.5447,-0.8327,0.0000
C01254=19.876,26.191,30.085,-175.2662,-26.2938,0.0000
C01255=20.863,24.802,29.771,-153.1710,-26.4641,0.0000
C01256=21.967,23.786,29.757,-150.3617,-24.2494,0.0000
C01257=22.894,22.894,29.766,-151.4532,-25.5414,0.0000
C01258=23.786,21.968,29.757,-152.6043,-26.8012,0.0000
C01259=24.802,20.862,29.771,-150.8441,-23.8286,0.0000
C01260=26.191,19.876,30.085,-153.6284,-4.2431,0.0000
C01261=27.638,20.163,30.880,-179.1673,0.4552,0.0000
C01262=29.482,21.332,31.987,176.6319,-2.1861,0.0000
C01263=31.823,23.028,33.135,174.8504,-3.5064,0.0000
C01264=34.442,24.946,34.017,173.6603,-4.2768,0.0000
C01265=36.982,26.615,34.453,172.9185,-2.9896,0.0000
C01266=39.714,26.951,34.683,175.2408,0.7662,0.0000
C01267=42.264,25.848,34.870,178.1183,1.4539,0.0000
C01268=44.106,23.511,35.059,179.9261,0.1362,0.0000
C01269=45.540,20.638,35.183,179.9923,0.0168,0.0000
C01270=46.795,17.608,35.183,179.9935,0.0173,0.0000
C01271=47.812,14.563,35.059,179.9559,0.1486,0.0000
C01272=48.163,11.608,34.870,-179.6978,2.3585,0.0000
C01273=47.139,9.024,34.683,-177.1730,3.9059,0.0000
C01274=44.970,7.331,34.453,-172.8718,2.8761,0.0000
C01275=41.994,6.715,34.017,-172.4936,1.4400,0.0000
C01276=38.785,6.219,33.135,-173.8797,1.1518,0.0000
C01277=35.931,5.763,31.987,-176.0726,0.8331,0.0000
C01278=33.800,5.286,30.880,179.0893,-0.2669,0.0000
C01279=32.574,4.465,30.085,163.7211,-21.4413,0.0000
C01280=32.290,2.786,29.771,177.8911,-36.9279,0.0000
C01281=32.352,1.286,29.757,-177.9468,-37.5348,0.0000
C01282=32.376,0.000,29.766,-179.9994,-37.5726,0.0000
C01283=32.352,-1.286,29.757,177.9461,-37.5348,0.0000
C01284=32.290,-2.786,29.771,-177.8883,-36.9273,0.0000
C01285=32.574,-4.465,30.085,-163.7212,-21.4413,0.0000
C01286=33.800,-5.286,30.880,-179.0893,-0.2669,0.0000
C01287=35.931,-5.763,31.987,176.0726,0.8331,0.0000
C01288=38.785,-6.219,33.135,173.8797,1.1518,0.0000
C01289=41.994,-6.715,34.017,172.4936,1.4400,0.0000
C01290=44.970,-7.331,34.453,172.8718,2.8761,0.0000
C01291=47.139,-9.024,34.683,177.1730,3.9059,0.0000
C01292=48.163,-11.608,34.870,179.6978,2.3585,0.0000
C01293=47.812,-14.563,35.059,-179.9559,0.1486,0.0000
C01294=46.795,-17.608,35.183,-179.9935,0.0173,0.0000
C01295=45.540,-20.638,35.183,-179.9923,0.0168,0.0000
C01296=44.106,-23.511,35.059,-179.9261,0.1362,0.0000
C01297=42.264,-25.848,34.870,-178.1183,1.4539,0.0000
C01298=39.714,-26.951,34.683,-175.2408,0.7662,0.0000
C01299=36.982,-26.615,34.453,-172.9185,-2.9896,0.0000
C01300=34.442,-24.946,34.017,-173.6603,-4.2768,0.0000
C01301=31.823,-23.028,33.135,-174.8504,-3.5064,0.0000
C01302=29.482,-21.332,31.987,-176.6319,-2.1861,0.0000
C01303=27.638,-20.163,30.880,179.1673,0.4552,0.0000
C01304=26.191,-19.876,30.085,153.6283,-4.2431,0.0000
C01305=24.802,-20.863,29.771,150.8451,-23.8307,0.0000
C01306=23.786,-21.967,29.757,152.6040,-26.8008,0.0000
C01307=22.894,-22.894,29.766,151.4539,-25.5422,0.0000
C01308=21.968,-23.786,29.757,150.3613,-24.2490,0.0000
C01309=20.862,-24.802,29.771,153.1730,-26.4655,0.0000
C01310=19.876,-26.191,30.085,175.2661,-26.2938,0.0000
C01311=20.163,-27.638,30.880,-179.5447,-0.8327,0.0000
C01312=21.332,-29.482,31.987,177.8101,3.3656,0.0000
C01313=23.028,-31.823,33.135,176.4794,5.1399,0.0000
C01314=24.946,-34.442,34.017,175.6970,6.3219,0.0000
C01315=26.615,-36.982,34.453,176.9875,7.0718,0.0000
C01316=26.951,-39.714,34.683,-179.2311,4.7588,0.0000
C01317=25.848,-42.264,34.870,-178.5453,1.8811,0.0000
C01318=23.511,-44.106,35.059,-179.8638,0.0739,0.0000
C01319=20.638,-45.540,35.183,-179.9832,0.0077,0.0000
C01320=17.608,-46.795,35.183,-179.9827,0.0065,0.0000
C01321=14.563,-47.812,35.059,-179.8514,0.0441,0.0000
C01322=11.608,-48.163,34.870,-177.6414,-0.3019,0.0000
C01323=9.024,-47.139,34.683,-176.0894,-2.8205,0.0000
C01324=7.331,-44.970,34.453,-177.1015,-7.1192,0.0000
C01325=6.715,-41.994,34.017,-178.5475,-7.5040,0.0000
C01326=6.219,-38.785,33.135,-178.8416,-6.1191,0.0000
C01327=5.763,-35.931,31.987,-179.1649,-3.9270,0.0000
C01328=5.286,-33.800,30.880,179.7331,0.9107,0.0000
C01329=4.465,-32.574,30.085,157.7490,15.1242,0.0000
C01330=2.786,-32.290,29.771,143.0534,1.6857,0.0000
C01331=1.286,-32.352,29.757,142.4475,-1.6281,0.0000
C01332=0.000,-32.376,29.766,142.4274,-0.0005,0.0000
C01333=0.000,-32.376,29.766,142.4274,-0.0005,0.0000
C01334=-1.286,-32.352,29.757,142.4474,1.6286,0.0000
C01335=-2.786,-32.290,29.771,143.0540,-1.6879,0.0000
C01336=-4.465,-32.574,30.085,157.7490,-15.1242,0.0000
C01337=-5.286,-33.800,30.880,179.7331,-0.9107,0.0000
C01338=-5.763,-35.931,31.987,-179.1649,3.9270,0.0000
C01339=-6.219,-38.785,33.135,-178.8416,6.1191,0.0000
C01340=-6.715,-41.994,34.017,-178.5475,7.5040,0.0000
C01341=-7.331,-44.970,34.453,-177.1015,7.1192,0.0000
C01342=-9.024,-47.139,34.683,-176.0894,2.8205,0.0000
C01343=-11.608,-48.163,34.870,-177.6414,0.3019,0.0000
C01344=-14.563,-47.812,35.059,-179.8514,-0.0441,0.0000
C01345=-17.608,-46.795,35.183,-179.9827,-0.0065,0.0000
C01346=-20.638,-45.540,35.183,-179.9832,-0.0077,0.0000
C01347=-23.511,-44.106,35.059,-179.8638,-0.0739,0.0000
C01348=-25.848,-42.264,34.870,-178.5453,-1.8811,0.0000
C01349=-26.951,-39.714,34.683,-179.2311,-4.7588,0.0000
C01350=-26.615,-36.982,34.453,176.9875,-7.0718,0.0000
C01351=-24.946,-34.442,34.017,175.6970,-6.3219,0.0000
C01352=-23.028,-31.823,33.135,176.4794,-5.1399,0.0000
C01353=-21.332,-29.482,31.987,177.8101,-3.3656,0.0000
C01354=-20.163,-27.638,30.880,-179.5447,0.8327,0.0000
C01355=-19.876,-26.191,30.085,175.2662,26.2938,0.0000
C01356=-20.863,-24.802,29.771,153.1710,26.4641,0.0000
C01357=-21.967,-23.786,29.757,150.3617,24.2494,0.0000
C01358=-22.894,-22.894,29.766,151.4532,25.5414,0.0000
C01359=-23.786,-21.968,29.757,152.6043,26.8012,0.0000
C01360=-24.802,-20.862,29.771,150.8441,23.8286,0.0000
C01361=-26.191,-19.876,30.085,153.6284,4.2431,0.0000
C01362=-27.638,-20.163,30.880,179.1673,-0.4552,0.0000
C01363=-29.482,-21.332,31.987,-176.6319,2.1861,0.0000
C01364=-31.823,-23.028,33.135,-174.8504,3.5064,0.0000
C01365=-34.442,-24.946,34.017,-173.6603,4.2768,0.0000
C01366=-36.982,-26.615,34.453,-172.9185,2.9896,0.0000
C01367=-39.714,-26.951,34.683,-175.2408,-0.7662,0.0000
C01368=-42.264,-25.848,34.870,-178.1183,-1.4539,0.0000
C01369=-44.106,-23.511,35.059,-179.9261,-0.1362,0.0000
C01370=-45.540,-20.638,35.183,-179.9923,-0.0168,0.0000
C01371=-46.795,-17.608,35.183,-179.9935,-0.0173,0.0000
C01372=-47.812,-14.563,35.059,-179.9559,-0.1486,0.0000
C01373=-48.163,-11.608,34.870,179.6978,-2.3585,0.0000
C01374=-47.139,-9.024,34.683,177.1730,-3.9059,0.0000
C01375=-44.970,-7.331,34.453,172.8718,-2.8761,0.0000
C01376=-41.994,-6.715,34.017,172.4936,-1.4400,0.0000
C01377=-38.785,-6.219,33.135,173.8797,-1.1518,0.0000
C01378=-35.931,-5.763,31.987,176.0726,-0.8331,0.0000
C01379=-33.800,-5.286,30.880,-179.0893,0.2669,0.0000
C01380=-32.574,-4.465,30.085,-163.7211,21.4413,0.0000
C01381=-32.290,-2.786,29.771,-177.8911,36.9279,0.0000
C01382=-32.352,-1.286,29.757,177.9468,37.5348,0.0000
C01383=-32.376,0.000,29.766,179.9994,37.5726,0.0000
C01384=-32.352,1.286,29.757,-177.9461,37.5348,0.0000
C01385=-32.290,2.786,29.771,177.8883,36.9273,0.0000
C01386=-32.574,4.465,30.085,163.7212,21.4413,0.0000
C01387=-33.800,5.286,30.880,179.0893,0.2669,0.0000
C01388=-35.931,5.763,31.987,-176.0726,-0.8331,0.0000
C01389=-38.785,6.219,33.135,-173.8797,-1.1518,0.0000
C01390=-41.994,6.715,34.017,-172.4936,-1.4400,0.0000
C01391=-44.970,7.331,34.453,-172.8718,-2.8761,0.0000
C01392=-47.139,9.024,34.683,-177.1730,-3.9059,0.0000
C01393=-48.163,11.608,34.870,-179.6978,-2.3585,0.0000
C01394=-47.812,14.563,35.059,179.9559,-0.1486,0.0000
C01395=-46.795,17.608,35.183,179.9935,-0.0173,0.0000
C01396=-45.540,20.638,35.183,179.9923,-0.0168,0.0000
C01397=-44.106,23.511,35.059,179.9261,-0.1362,0.0000
C01398=-42.264,25.848,34.870,178.1183,-1.4539,0.0000
C01399=-39.714,26.951,34.683,175.2408,-0.7662,0.0000
C01400=-36.982,26.615,34.453,172.9185,2.9896,0.0000
C01401=-34.442,24.946,34.017,173.6603,4.2768,0.0000
C01402=-31.823,23.028,33.135,174.8504,3.5064,0.0000
C01403=-29.482,21.332,31.987,176.6319,2.1861,0.0000
C01404=-27.638,20.163,30.880,-179.1673,-0.4552,0.0000
C01405=-26.191,19.876,30.085,-153.6283,4.2431,0.0000
C01406=-24.802,20.863,29.771,-150.8451,23.8307,0.0000
C01407=-23.786,21.967,29.757,-152.6040,26.8008,0.0000
C01408=-22.894,22.894,29.766,-151.4539,25.5422,0.0000
C01409=-21.968,23.786,29.757,-150.3613,24.2490,0.0000
C01410=-20.862,24.802,29.771,-153.1730,26.4655,0.0000
C01411=-19.876,26.191,30.085,-175.2661,26.2938,0.0000
C01412=-20.163,27.638,30.880,179.5447,0.8327,0.0000
C01413=-21.332,29.482,31.987,-177.8101,-3.3656,0.0000
C01414=-23.028,31.823,33.135,-176.4794,-5.1399,0.0000
C01415=-24.946,34.442,34.017,-175.6970,-6.3219,0.0000
C01416=-26.615,36.982,34.453,-176.9875,-7.0718,0.0000
C01417=-26.951,39.714,34.683,179.2311,-4.7588,0.0000
C01418=-25.848,42.264,34.870,178.5453,-1.8811,0.0000
C01419=-23.511,44.106,35.059,179.8638,-0.0739,0.0000
C01420=-20.638,45.540,35.183,179.9832,-0.0077,0.0000
C01421=-17.608,46.795,35.183,179.9827,-0.0065,0.0000
C01422=-14.563,47.812,35.059,179.8514,-0.0441,0.0000
C01423=-11.608,48.163,34.870,177.6414,0.3019,0.0000
C01424=-9.024,47.139,34.683,176.0894,2.8205,0.0000
C01425=-7.331,44.970,34.453,177.1015,7.1192,0.0000
C01426=-6.715,41.994,34.017,178.5475,7.5040,0.0000
C01427=-6.219,38.785,33.135,178.8416,6.1191,0.0000
C01428=-5.763,35.931,31.987,179.1649,3.9270,0.0000
C01429=-5.286,33.800,30.880,-179.7331,-0.9107,0.0000
C01430=-4.465,32.574,30.085,-157.7490,-15.1242,0.0000
C01431=-2.786,32.290,29.771,-143.0540,-1.6879,0.0000
C01432=-1.286,32.352,29.757,-142.4474,1.6286,0.0000
C01433=0.000,32.376,29.766,-142.4274,-0.0005,0.0000
C01434=0.000,31.053,31.524,-143.6768,-0.0006,0.0000
C01435=1.165,31.033,31.514,-143.6940,-1.5129,0.0000
C01436=2.582,30.983,31.529,-144.4304,2.2364,0.0000
C01437=4.218,31.318,31.874,-160.6310,14.8582,0.0000
C01438=4.987,32.673,32.745,179.9109,-0.3504,0.0000
C01439=5.430,35.005,33.954,179.1939,-4.2040,0.0000
C01440=5.871,38.106,35.198,178.9774,-5.9064,0.0000
C01441=6.356,41.567,36.145,178.7757,-7.0003,0.0000
C01442=6.949,44.762,36.610,177.5058,-6.6410,0.0000
C01443=8.669,47.097,36.854,176.4306,-2.7166,0.0000
C01444=11.329,48.213,37.052,177.8254,-0.3084,0.0000
C01445=14.389,47.870,37.251,179.8617,0.0408,0.0000
C01446=17.550,46.817,37.382,179.9840,0.0060,0.0000
C01447=20.695,45.514,37.382,179.9845,0.0071,0.0000
C01448=23.675,44.023,37.251,179.8733,0.0690,0.0000
C01449=26.081,42.103,37.052,178.6800,1.7556,0.0000
C01450=27.172,39.432,36.854,179.3989,4.4441,0.0000
C01451=26.738,36.565,36.610,-177.0459,6.4503,0.0000
C01452=24.898,33.886,36.145,-175.8970,5.8067,0.0000
C01453=22.793,31.096,35.198,-176.5354,4.8942,0.0000
C01454=20.912,28.592,33.954,-177.5931,3.5407,0.0000
C01455=19.577,26.630,32.745,-179.8152,0.3107,0.0000
C01456=19.163,25.127,31.874,-177.1528,-24.0788,0.0000
C01457=20.082,23.734,31.529,-154.7457,-26.0144,0.0000
C01458=21.120,22.768,31.514,-151.5108,-23.5695,0.0000
C01459=21.958,21.958,31.524,-152.5313,-24.7613,0.0000
C01460=22.768,21.120,31.514,-153.6024,-25.9259,0.0000
C01461=23.734,20.082,31.529,-151.6468,-22.5429,0.0000
C01462=25.127,19.163,31.874,-155.8950,-2.5991,0.0000
C01463=26.630,19.577,32.745,179.6893,-0.1848,0.0000
C01464=28.592,20.912,33.954,176.4562,-2.4023,0.0000
C01465=31.096,22.793,35.198,175.0969,-3.4520,0.0000
C01466=33.886,24.898,36.145,174.1785,-4.0819,0.0000
C01467=36.565,26.738,36.610,173.5411,-2.9354,0.0000
C01468=39.432,27.172,36.854,175.5556,0.5993,0.0000
C01469=42.103,26.081,37.052,178.2439,1.3193,0.0000
C01470=44.023,23.675,37.251,179.9310,0.1267,0.0000
C01471=45.514,20.695,37.382,179.9929,0.0155,0.0000
C01472=46.817,17.550,37.382,179.9940,0.0160,0.0000
C01473=47.870,14.389,37.251,179.9592,0.1383,0.0000
C01474=48.213,11.329,37.052,-179.6914,2.1746,0.0000
C01475=47.097,8.669,36.854,-177.2782,3.5654,0.0000
C01476=44.762,6.949,36.610,-173.3527,2.4775,0.0000
C01477=41.567,6.356,36.145,-172.9982,1.2151,0.0000
C01478=38.106,5.871,35.198,-174.0927,1.0171,0.0000
C01479=35.005,5.430,33.954,-175.7956,0.8039,0.0000
C01480=32.673,4.987,32.745,-179.6496,0.0890,0.0000
C01481=31.318,4.218,31.874,164.2933,-18.6969,0.0000
C01482=30.983,2.582,31.529,177.2513,-35.5384,0.0000
C01483=31.033,1.165,31.514,-178.1229,-36.2914,0.0000
C01484=31.053,0.000,31.524,-179.9992,-36.3232,0.0000
C01485=31.033,-1.165,31.514,178.1220,-36.2914,0.0000
C01486=30.983,-2.582,31.529,-177.2485,-35.5377,0.0000
C01487=31.318,-4.218,31.874,-164.2933,-18.6967,0.0000
C01488=32.673,-4.987,32.745,179.6496,0.0890,0.0000
C01489=35.005,-5.430,33.954,175.7956,0.8039,0.0000
C01490=38.106,-5.871,35.198,174.0927,1.0171,0.0000
C01491=41.567,-6.356,36.145,172.9982,1.2151,0.0000
C01492=44.762,-6.949,36.610,173.3527,2.4775,0.0000
C01493=47.097,-8.669,36.854,177.2782,3.5654,0.0000
C01494=48.213,-11.329,37.052,179.6914,2.1746,0.0000
C01495=47.870,-14.389,37.251,-179.9592,0.1383,0.0000
C01496=46.817,-17.550,37.382,-179.9940,0.0160,0.0000
C01497=45.514,-20.695,37.382,-179.9929,0.0155,0.0000
C01498=44.023,-23.675,37.251,-179.9310,0.1267,0.0000
C01499=42.103,-26.081,37.052,-178.2439,1.3193,0.0000
C01500=39.432,-27.172,36.854,-175.5556,0.5993,0.0000
C01501=36.565,-26.738,36.610,-173.5411,-2.9354,0.0000
C01502=33.886,-24.898,36.145,-174.1785,-4.0819,0.0000
C01503=31.096,-22.793,35.198,-175.0969,-3.4520,0.0000
C01504=28.592,-20.912,33.954,-176.4562,-2.4023,0.0000
C01505=26.630,-19.577,32.745,-179.6893,-0.1848,0.0000
C01506=25.127,-19.163,31.874,155.8948,-2.5992,0.0000
C01507=23.734,-20.082,31.529,151.6478,-22.5451,0.0000
C01508=22.768,-21.120,31.514,153.6019,-25.9253,0.0000
C01509=21.958,-21.958,31.524,152.5322,-24.7623,0.0000
C01510=21.120,-22.768,31.514,151.5104,-23.5690,0.0000
C01511=20.082,-23.734,31.529,154.7479,-26.0158,0.0000
C01512=19.163,-25.127,31.874,177.1530,-24.0787,0.0000
C01513=19.577,-26.630,32.745,179.8152,0.3107,0.0000
C01514=20.912,-28.592,33.954,177.5931,3.5407,0.0000
C01515=22.793,-31.096,35.198,176.5354,4.8942,0.0000
C01516=24.898,-33.886,36.145,175.8970,5.8067,0.0000
C01517=26.738,-36.565,36.610,177.0459,6.4503,0.0000
C01518=27.172,-39.432,36.854,-179.3989,4.4441,0.0000
C01519=26.081,-42.103,37.052,-178.6800,1.7556,0.0000
C01520=23.675,-44.023,37.251,-179.8733,0.0690,0.0000
C01521=20.695,-45.514,37.382,-179.9845,0.0071,0.0000
C01522=17.550,-46.817,37.382,-179.9840,0.0060,0.0000
C01523=14.389,-47.870,37.251,-179.8617,0.0408,0.0000
C01524=11.329,-48.213,37.052,-177.8254,-0.3084,0.0000
C01525=8.669,-47.097,36.854,-176.4306,-2.7166,0.0000
C01526=6.949,-44.762,36.610,-177.5058,-6.6410,0.0000
C01527=6.356,-41.567,36.145,-178.7757,-7.0003,0.0000
C01528=5.871,-38.106,35.198,-178.9774,-5.9064,0.0000
C01529=5.430,-35.005,33.954,-179.1939,-4.2040,0.0000
C01530=4.987,-32.673,32.745,-179.9109,-0.3504,0.0000
C01531=4.218,-31.318,31.874,160.6310,14.8582,0.0000
C01532=2.582,-30.983,31.529,144.4304,2.2364,0.0000
C01533=1.165,-31.033,31.514,143.6940,-1.5129,0.0000
C01534=0.000,-31.053,31.524,143.6768,-0.0006,0.0000
C01535=0.000,-31.053,31.524,143.6768,-0.0006,0.0000
C01536=-1.165,-31.033,31.514,143.6939,1.5136,0.0000
C01537=-2.582,-30.983,31.529,144.4311,-2.2387,0.0000
C01538=-4.218,-31.318,31.874,160.6312,-14.8582,0.0000
C01539=-4.987,-32.673,32.745,-179.9109,0.3504,0.0000
C01540=-5.430,-35.005,33.954,-179.1939,4.2040,0.0000
C01541=-5.871,-38.106,35.198,-178.9774,5.9064,0.0000
C01542=-6.356,-41.567,36.145,-178.7757,7.0003,0.0000
C01543=-6.949,-44.762,36.610,-177.5058,6.6410,0.0000
C01544=-8.669,-47.097,36.854,-176.4306,2.7166,0.0000
C01545=-11.329,-48.213,37.052,-177.8254,0.3084,0.0000
C01546=-14.389,-47.870,37.251,-179.8617,-0.0408,0.0000
C01547=-17.550,-46.817,37.382,-179.9840,-0.0060,0.0000
C01548=-20.695,-45.514,37.382,-179.9845,-0.0071,0.0000
C01549=-23.675,-44.023,37.251,-179.8733,-0.0690,0.0000
C01550=-26.081,-42.103,37.052,-178.6800,-1.7556,0.0000
C01551=-27.172,-39.432,36.854,-179.3989,-4.4441,0.0000
C01552=-26.738,-36.565,36.610,177.0459,-6.4503,0.0000
C01553=-24.898,-33.886,36.145,175.8970,-5.8067,0.0000
C01554=-22.793,-31.096,35.198,176.5354,-4.8942,0.0000
C01555=-20.912,-28.592,33.954,177.5931,-3.5407,0.0000
C01556=-19.577,-26.630,32.745,179.8152,-0.3107,0.0000
C01557=-19.163,-25.127,31.874,177.1528,24.0788,0.0000
C01558=-20.082,-23.734,31.529,154.7457,26.0144,0.0000
C01559=-21.120,-22.768,31.514,151.5108,23.5695,0.0000
C01560=-21.958,-21.958,31.524,152.5313,24.7613,0.0000
C01561=-22.768,-21.120,31.514,153.6024,25.9259,0.0000
C01562=-23.734,-20.082,31.529,151.6468,22.5429,0.0000
C01563=-25.127,-19.163,31.874,155.8950,2.5991,0.0000
C01564=-26.630,-19.577,32.745,-179.6893,0.1848,0.0000
C01565=-28.592,-20.912,33.954,-176.4562,2.4023,0.0000
C01566=-31.096,-22.793,35.198,-175.0969,3.4520,0.0000
C01567=-33.886,-24.898,36.145,-174.1785,4.0819,0.0000
C01568=-36.565,-26.738,36.610,-173.5411,2.9354,0.0000
C01569=-39.432,-27.172,36.854,-175.5556,-0.5993,0.0000
C01570=-42.103,-26.081,37.052,-178.2439,-1.3193,0.0000
C01571=-44.023,-23.675,37.251,-179.9310,-0.1267,0.0000
C01572=-45.514,-20.695,37.382,-179.9929,-0.0155,0.0000
C01573=-46.817,-17.550,37.382,-179.9940,-0.0160,0.0000
C01574=-47.870,-14.389,37.251,-179.9592,-0.1383,0.0000
C01575=-48.213,-11.329,37.052,179.6914,-2.1746,0.0000
C01576=-47.097,-8.669,36.854,177.2782,-3.5654,0.0000
C01577=-44.762,-6.949,36.610,173.3527,-2.4775,0.0000
C01578=-41.567,-6.356,36.145,172.9982,-1.2151,0.0000
C01579=-38.106,-5.871,35.198,174.0927,-1.0171,0.0000
C01580=-35.005,-5.430,33.954,175.7956,-0.8039,0.0000
C01581=-32.673,-4.987,32.745,179.6496,-0.0890,0.0000
C01582=-31.318,-4.218,31.874,-164.2933,18.6969,0.0000
C01583=-30.983,-2.582,31.529,-177.2513,35.5384,0.0000
C01584=-31.033,-1.165,31.514,178.1229,36.2914,0.0000
C01585=-31.053,0.000,31.524,179.9992,36.3232,0.0000
C01586=-31.033,1.165,31.514,-178.1220,36.2914,0.0000
C01587=-30.983,2.582,31.529,177.2485,35.5377,0.0000
C01588=-31.318,4.218,31.874,164.2933,18.6967,0.0000
C01589=-32.673,4.987,32.745,-179.6496,-0.0890,0.0000
C01590=-35.005,5.430,33.954,-175.7956,-0.8039,0.0000
C01591=-38.106,5.871,35.198,-174.0927,-1.0171,0.0000
C01592=-41.567,6.356,36.145,-172.9982,-1.2151,0.0000
C01593=-44.762,6.949,36.610,-173.3527,-2.4775,0.0000
C01594=-47.097,8.669,36.854,-177.2782,-3.5654,0.0000
C01595=-48.213,11.329,37.052,-179.6914,-2.1746,0.0000
C01596=-47.870,14.389,37.251,179.9592,-0.1383,0.0000
C01597=-46.817,17.550,37.382,179.9940,-0.0160,0.0000
C01598=-45.514,20.695,37.382,179.9929,-0.0155,0.0000
C01599=-44.023,23.675,37.251,179.9310,-0.1267,0.0000
C01600=-42.103,26.081,37.052,178.2439,-1.3193,0.0000
C01601=-39.432,27.172,36.854,175.5556,-0.5993,0.0000
C01602=-36.565,26.738,36.610,173.5411,2.9354,0.0000
C01603=-33.886,24.898,36.145,174.1785,4.0819,0.0000
C01604=-31.096,22.793,35.198,175.0969,3.4520,0.0000
C01605=-28.592,20.912,33.954,176.4562,2.4023,0.0000
C01606=-26.630,19.577,32.745,179.6893,0.1848,0.0000
C01607=-25.127,19.163,31.874,-155.8948,2.5992,0.0000
C01608=-23.734,20.082,31.529,-151.6478,22.5451,0.0000
C01609=-22.768,21.120,31.514,-153.6019,25.9253,0.0000
C01610=-21.958,21.958,31.524,-152.5322,24.7623,0.0000
C01611=-21.120,22.768,31.514,-151.5104,23.5690,0.0000
C01612=-20.082,23.734,31.529,-154.7479,26.0158,0.0000
C01613=-19.163,25.127,31.874,-177.1530,24.0787,0.0000
C01614=-19.577,26.630,32.745,-179.8152,-0.3107,0.0000
C01615=-20.912,28.592,33.954,-177.5931,-3.5407,0.0000
C01616=-22.793,31.096,35.198,-176.5354,-4.8942,0.0000
C01617=-24.898,33.886,36.145,-175.8970,-5.8067,0.0000
C01618=-26.738,36.565,36.610,-177.0459,-6.4503,0.0000
C01619=-27.172,39.432,36.854,179.3989,-4.4441,0.0000
C01620=-26.081,42.103,37.052,178.6800,-1.7556,0.0000
C01621=-23.675,44.023,37.251,179.8733,-0.0690,0.0000
C01622=-20.695,45.514,37.382,179.9845,-0.0071,0.0000
C01623=-17.550,46.817,37.382,179.9840,-0.0060,0.0000
C01624=-14.389,47.870,37.251,179.8617,-0.0408,0.0000
C01625=-11.329,48.213,37.052,177.8254,0.3084,0.0000
C01626=-8.669,47.097,36.854,176.4306,2.7166,0.0000
C01627=-6.949,44.762,36.610,177.5058,6.6410,0.0000
C01628=-6.356,41.567,36.145,178.7757,7.0003,0.0000
C01629=-5.871,38.106,35.198,178.9774,5.9064,0.0000
C01630=-5.430,35.005,33.954,179.1939,4.2040,0.0000
C01631=-4.987,32.673,32.745,179.9109,0.3504,0.0000
C01632=-4.218,31.318,31.874,-160.6312,-14.8582,0.0000
C01633=-2.582,30.983,31.529,-144.4311,-2.2387,0.0000
C01634=-1.165,31.033,31.514,-143.6939,1.5136,0.0000
C01635=0.000,31.053,31.524,-143.6768,-0.0006,0.0000
C01636=0.000,29.775,33.314,-145.3452,-0.0007,0.0000
C01637=1.048,29.759,33.303,-145.3590,-1.3756,0.0000
C01638=2.386,29.720,33.319,-146.2392,2.7343,0.0000
C01639=3.979,30.109,33.696,-163.5073,14.1247,0.0000
C01640=4.702,31.601,34.645,179.7169,-1.2741,0.0000
C01641=5.119,34.140,35.953,179.2621,-4.2246,0.0000
C01642=5.555,37.486,37.285,179.1265,-5.4560,0.0000
C01643=6.036,41.186,38.288,179.0008,-6.2396,0.0000
C01644=6.613,44.579,38.776,177.9344,-5.8850,0.0000
C01645=8.359,47.059,39.032,176.9019,-2.4616,0.0000
C01646=11.087,48.257,39.238,178.0988,-0.2912,0.0000
C01647=14.238,47.919,39.446,179.8785,0.0356,0.0000
C01648=17.499,46.837,39.582,179.9861,0.0052,0.0000
C01649=20.745,45.492,39.582,179.9865,0.0062,0.0000
C01650=23.816,43.952,39.446,179.8889,0.0607,0.0000
C01651=26.283,41.963,39.238,178.8613,1.5501,0.0000
C01652=27.365,39.186,39.032,179.5514,3.9308,0.0000
C01653=26.846,36.198,38.776,-177.2845,5.6156,0.0000
C01654=24.854,33.391,38.288,-176.2815,5.1124,0.0000
C01655=22.579,30.435,37.285,-176.7511,4.4716,0.0000
C01656=20.521,27.760,35.953,-177.5304,3.5070,0.0000
C01657=19.020,25.670,34.645,-179.2991,1.1011,0.0000
C01658=18.476,24.104,33.696,-178.6375,-21.5450,0.0000
C01659=19.328,22.702,33.319,-156.6335,-25.2294,0.0000
C01660=20.302,21.784,33.303,-153.0154,-22.6346,0.0000
C01661=21.054,21.054,33.314,-153.9502,-23.7079,0.0000
C01662=21.784,20.302,33.303,-154.9252,-24.7596,0.0000
C01663=22.702,19.328,33.320,-152.8282,-21.0229,0.0000
C01664=24.104,18.476,33.696,-158.4498,-1.2670,0.0000
C01665=25.670,19.020,34.645,178.8988,-0.7007,0.0000
C01666=27.760,20.521,35.953,176.4897,-2.4650,0.0000
C01667=30.435,22.579,37.285,175.5213,-3.2390,0.0000
C01668=33.391,24.854,38.288,174.8768,-3.7036,0.0000
C01669=36.198,26.846,38.776,174.3781,-2.7025,0.0000
C01670=39.186,27.365,39.032,176.0691,0.4475,0.0000
C01671=41.963,26.283,39.238,178.4496,1.1383,0.0000
C01672=43.952,23.816,39.446,179.9393,0.1111,0.0000
C01673=45.492,20.745,39.582,179.9938,0.0135,0.0000
C01674=46.837,17.499,39.582,179.9948,0.0139,0.0000
C01675=47.919,14.238,39.446,179.9644,0.1215,0.0000
C01676=48.257,11.087,39.238,-179.7087,1.9011,0.0000
C01677=47.059,8.359,39.032,-177.5348,3.0952,0.0000
C01678=44.579,6.613,38.776,-174.1112,2.0547,0.0000
C01679=41.186,6.036,38.288,-173.7594,0.9932,0.0000
C01680=37.486,5.555,37.285,-174.5434,0.8696,0.0000
C01681=34.140,5.119,35.953,-175.7751,0.7359,0.0000
C01682=31.601,4.702,34.645,-178.7259,0.2830,0.0000
C01683=30.109,3.979,33.696,165.2950,-15.9805,0.0000
C01684=29.720,2.386,33.319,176.7121,-33.7172,0.0000
C01685=29.759,1.048,33.303,-178.3282,-34.6296,0.0000
C01686=29.775,0.000,33.314,-179.9991,-34.6548,0.0000
C01687=29.759,-1.048,33.303,178.3272,-34.6297,0.0000
C01688=29.720,-2.386,33.320,-176.7094,-33.7164,0.0000
C01689=30.109,-3.979,33.696,-165.2950,-15.9801,0.0000
C01690=31.601,-4.702,34.645,178.7259,0.2830,0.0000
C01691=34.140,-5.119,35.953,175.7751,0.7359,0.0000
C01692=37.486,-5.555,37.285,174.5434,0.8696,0.0000
C01693=41.186,-6.036,38.288,173.7594,0.9932,0.0000
C01694=44.579,-6.613,38.776,174.1112,2.0547,0.0000
C01695=47.059,-8.359,39.032,177.5348,3.0952,0.0000
C01696=48.257,-11.087,39.238,179.7087,1.9011,0.0000
C01697=47.919,-14.238,39.446,-179.9644,0.1215,0.0000
C01698=46.837,-17.499,39.582,-179.9948,0.0139,0.0000
C01699=45.492,-20.745,39.582,-179.9938,0.0135,0.0000
C01700=43.952,-23.816,39.446,-179.9393,0.1111,0.0000
C01701=41.963,-26.283,39.238,-178.4496,1.1383,0.0000
C01702=39.186,-27.365,39.032,-176.0691,0.4475,0.0000
C01703=36.198,-26.846,38.776,-174.3781,-2.7025,0.0000
C01704=33.391,-24.854,38.288,-174.8768,-3.7036,0.0000
C01705=30.435,-22.579,37.285,-175.5213,-3.2390,0.0000
C01706=27.760,-20.521,35.953,-176.4897,-2.4650,0.0000
C01707=25.670,-19.020,34.645,-178.8988,-0.7007,0.0000
C01708=24.104,-18.476,33.696,158.4495,-1.2673,0.0000
C01709=22.702,-19.328,33.319,152.8291,-21.0252,0.0000
C01710=21.784,-20.302,33.303,154.9246,-24.7590,0.0000
C01711=21.054,-21.054,33.314,153.9512,-23.7090,0.0000
C01712=20.302,-21.784,33.303,153.0148,-22.6340,0.0000
C01713=19.328,-22.702,33.320,156.6358,-25.2307,0.0000
C01714=18.476,-24.104,33.696,178.6378,-21.5446,0.0000
C01715=19.020,-25.670,34.645,179.2991,1.1011,0.0000
C01716=20.521,-27.760,35.953,177.5304,3.5070,0.0000
C01717=22.579,-30.435,37.285,176.7511,4.4716,0.0000
C01718=24.854,-33.391,38.288,176.2815,5.1124,0.0000
C01719=26.846,-36.198,38.776,177.2845,5.6156,0.0000
C01720=27.365,-39.186,39.032,-179.5514,3.9308,0.0000
C01721=26.283,-41.963,39.238,-178.8613,1.5501,0.0000
C01722=23.816,-43.952,39.446,-179.8889,0.0607,0.0000
C01723=20.745,-45.492,39.582,-179.9865,0.0062,0.0000
C01724=17.499,-46.837,39.582,-179.9861,0.0052,0.0000
C01725=14.238,-47.919,39.446,-179.8785,0.0356,0.0000
C01726=11.087,-48.257,39.238,-178.0988,-0.2912,0.0000
C01727=8.359,-47.059,39.032,-176.9019,-2.4616,0.0000
C01728=6.613,-44.579,38.776,-177.9344,-5.8850,0.0000
C01729=6.036,-41.186,38.288,-179.0008,-6.2396,0.0000
C01730=5.555,-37.486,37.285,-179.1265,-5.4560,0.0000
C01731=5.119,-34.140,35.953,-179.2621,-4.2246,0.0000
C01732=4.702,-31.601,34.645,-179.7169,-1.2741,0.0000
C01733=3.979,-30.109,33.696,163.5073,14.1247,0.0000
C01734=2.386,-29.720,33.319,146.2392,2.7343,0.0000
C01735=1.048,-29.759,33.303,145.3590,-1.3756,0.0000
C01736=0.000,-29.775,33.314,145.3452,-0.0007,0.0000
C01737=0.000,-29.775,33.314,145.3452,-0.0007,0.0000
C01738=-1.048,-29.759,33.303,145.3589,1.3764,0.0000
C01739=-2.386,-29.720,33.320,146.2399,-2.7367,0.0000
C01740=-3.979,-30.109,33.696,163.5077,-14.1247,0.0000
C01741=-4.702,-31.601,34.645,-179.7169,1.2741,0.0000
C01742=-5.119,-34.140,35.953,-179.2621,4.2246,0.0000
C01743=-5.555,-37.486,37.285,-179.1265,5.4560,0.0000
C01744=-6.036,-41.186,38.288,-179.0008,6.2396,0.0000
C01745=-6.613,-44.579,38.776,-177.9344,5.8850,0.0000
C01746=-8.359,-47.059,39.032,-176.9019,2.4616,0.0000
C01747=-11.087,-48.257,39.238,-178.0988,0.2912,0.0000
C01748=-14.238,-47.919,39.446,-179.8785,-0.0356,0.0000
C01749=-17.499,-46.837,39.582,-179.9861,-0.0052,0.0000
C01750=-20.745,-45.492,39.582,-179.9865,-0.0062,0.0000
C01751=-23.816,-43.952,39.446,-179.8889,-0.0607,0.0000
C01752=-26.283,-41.963,39.238,-178.8613,-1.5501,0.0000
C01753=-27.365,-39.186,39.032,-179.5514,-3.9308,0.0000
C01754=-26.846,-36.198,38.776,177.2845,-5.6156,0.0000
C01755=-24.854,-33.391,38.288,176.2815,-5.1124,0.0000
C01756=-22.579,-30.435,37.285,176.7511,-4.4716,0.0000
C01757=-20.521,-27.760,35.953,177.5304,-3.5070,0.0000
C01758=-19.020,-25.670,34.645,179.2991,-1.1011,0.0000
C01759=-18.476,-24.104,33.696,178.6375,21.5450,0.0000
C01760=-19.328,-22.702,33.319,156.6335,25.2294,0.0000
C01761=-20.302,-21.784,33.303,153.0154,22.6346,0.0000
C01762=-21.054,-21.054,33.314,153.9502,23.7079,0.0000
C01763=-21.784,-20.302,33.303,154.9252,24.7596,0.0000
C01764=-22.702,-19.328,33.320,152.8282,21.0229,0.0000
C01765=-24.104,-18.476,33.696,158.4498,1.2670,0.0000
C01766=-25.670,-19.020,34.645,-178.8988,0.7007,0.0000
C01767=-27.760,-20.521,35.953,-176.4897,2.4650,0.0000
C01768=-30.435,-22.579,37.285,-175.5213,3.2390,0.0000
C01769=-33.391,-24.854,38.288,-174.8768,3.7036,0.0000
C01770=-36.198,-26.846,38.776,-174.3781,2.7025,0.0000
C01771=-39.186,-27.365,39.032,-176.0691,-0.4475,0.0000
C01772=-41.963,-26.283,39.238,-178.4496,-1.1383,0.0000
C01773=-43.952,-23.816,39.446,-179.9393,-0.1111,0.0000
C01774=-45.492,-20.745,39.582,-179.9938,-0.0135,0.0000
C01775=-46.837,-17.499,39.582,-179.9948,-0.0139,0.0000
C01776=-47.919,-14.238,39.446,-179.9644,-0.1215,0.0000
C01777=-48.257,-11.087,39.238,179.7087,-1.9011,0.0000
C01778=-47.059,-8.359,39.032,177.5348,-3.0952,0.0000
C01779=-44.579,-6.613,38.776,174.1112,-2.0547,0.0000
C01780=-41.186,-6.036,38.288,173.7594,-0.9932,0.0000
C01781=-37.486,-5.555,37.285,174.5434,-0.8696,0.0000
C01782=-34.140,-5.119,35.953,175.7751,-0.7359,0.0000
C01783=-31.601,-4.702,34.645,178.7259,-0.2830,0.0000
C01784=-30.109,-3.979,33.696,-165.2950,15.9805,0.0000
C01785=-29.720,-2.386,33.319,-176.7121,33.7172,0.0000
C01786=-29.759,-1.048,33.303,178.3282,34.6296,0.0000
C01787=-29.775,0.000,33.314,179.9991,34.6548,0.0000
C01788=-29.759,1.048,33.303,-178.3272,34.6297,0.0000
C01789=-29.720,2.386,33.320,176.7094,33.7164,0.0000
C01790=-30.109,3.979,33.696,165.2950,15.9801,0.0000
C01791=-31.601,4.702,34.645,-178.7259,-0.2830,0.0000
C01792=-34.140,5.119,35.953,-175.7751,-0.7359,0.0000
C01793=-37.486,5.555,37.285,-174.5434,-0.8696,0.0000
C01794=-41.186,6.036,38.288,-173.7594,-0.9932,0.0000
C01795=-44.579,6.613,38.776,-174.1112,-2.0547,0.0000
C01796=-47.059,8.359,39.032,-177.5348,-3.0952,0.0000
C01797=-48.257,11.087,39.238,-179.7087,-1.9011,0.0000
C01798=-47.919,14.238,39.446,179.9644,-0.1215,0.0000
C01799=-46.837,17.499,39.582,179.9948,-0.0139,0.0000
C01800=-45.492,20.745,39.582,179.9938,-0.0135,0.0000
C01801=-43.952,23.816,39.446,179.9393,-0.1111,0.0000
C01802=-41.963,26.283,39.238,178.4496,-1.1383,0.0000
C01803=-39.186,27.365,39.032,176.0691,-0.4475,0.0000
C01804=-36.198,26.846,38.776,174.3781,2.7025,0.0000
C01805=-33.391,24.854,38.288,174.8768,3.7036,0.0000
C01806=-30.435,22.579,37.285,175.5213,3.2390,0.0000
C01807=-27.760,20.521,35.953,176.4897,2.4650,0.0000
C01808=-25.670,19.020,34.645,178.8988,0.7007,0.0000
C01809=-24.104,18.476,33.696,-158.4495,1.2673,0.0000
C01810=-22.702,19.328,33.319,-152.8291,21.0252,0.0000
C01811=-21.784,20.302,33.303,-154.9246,24.7590,0.0000
C01812=-21.054,21.054,33.314,-153.9512,23.7090,0.0000
C01813=-20.302,21.784,33.303,-153.0148,22.6340,0.0000
C01814=-19.328,22.702,33.320,-156.6358,25.2307,0.0000
C01815=-18.476,24.104,33.696,-178.6378,21.5446,0.0000
C01816=-19.020,25.670,34.645,-179.2991,-1.1011,0.0000
C01817=-20.521,27.760,35.953,-177.5304,-3.5070,0.0000
C01818=-22.579,30.435,37.285,-176.7511,-4.4716,0.0000
C01819=-24.854,33.391,38.288,-176.2815,-5.1124,0.0000
C01820=-26.846,36.198,38.776,-177.2845,-5.6156,0.0000
C01821=-27.365,39.186,39.032,179.5514,-3.9308,0.0000
C01822=-26.283,41.963,39.238,178.8613,-1.5501,0.0000
C01823=-23.816,43.952,39.446,179.8889,-0.0607,0.0000
C01824=-20.745,45.492,39.582,179.9865,-0.0062,0.0000
C01825=-17.499,46.837,39.582,179.9861,-0.0052,0.0000
C01826=-14.238,47.919,39.446,179.8785,-0.0356,0.0000
C01827=-11.087,48.257,39.238,178.0988,0.2912,0.0000
C01828=-8.359,47.059,39.032,176.9019,2.4616,0.0000
C01829=-6.613,44.579,38.776,177.9344,5.8850,0.0000
C01830=-6.036,41.186,38.288,179.0008,6.2396,0.0000
C01831=-5.555,37.486,37.285,179.1265,5.4560,0.0000
C01832=-5.119,34.140,35.953,179.2621,4.2246,0.0000
C01833=-4.702,31.601,34.645,179.7169,1.2741,0.0000
C01834=-3.979,30.109,33.696,-163.5077,-14.1247,0.0000
C01835=-2.386,29.720,33.320,-146.2399,-2.7367,0.0000
C01836=-1.048,29.759,33.303,-145.3589,1.3764,0.0000
C01837=0.000,29.775,33.314,-145.3452,-0.0007,0.0000
C01838=0.000,28.557,35.146,-147.5083,-0.0008,0.0000
C01839=0.937,28.545,35.134,-147.5179,-1.2153,0.0000
C01840=2.198,28.517,35.152,-148.5454,3.1396,0.0000
C01841=3.753,28.963,35.561,-166.2907,12.9687,0.0000
C01842=4.437,30.601,36.587,179.6344,-1.8654,0.0000
C01843=4.837,33.354,37.988,179.3571,-3.9980,0.0000
C01844=5.276,36.942,39.399,179.2849,-4.7747,0.0000
C01845=5.763,40.861,40.447,179.2220,-5.2308,0.0000
C01846=6.331,44.425,40.953,178.3833,-4.8651,0.0000
C01847=8.101,47.028,41.216,177.4938,-2.0588,0.0000
C01848=10.888,48.294,41.429,178.4590,-0.2497,0.0000
C01849=14.116,47.960,41.642,179.9017,0.0287,0.0000
C01850=17.458,46.852,41.781,179.9888,0.0041,0.0000
C01851=20.785,45.474,41.781,179.9892,0.0050,0.0000
C01852=23.932,43.894,41.642,179.9101,0.0492,0.0000
C01853=26.450,41.848,41.429,179.0868,1.2662,0.0000
C01854=27.526,38.982,41.216,179.6845,3.2276,0.0000
C01855=26.937,35.890,40.953,-177.6949,4.5798,0.0000
C01856=24.818,32.968,40.447,-176.8439,4.2453,0.0000
C01857=22.391,29.853,39.399,-177.1238,3.8792,0.0000
C01858=20.165,27.005,37.988,-177.6242,3.2800,0.0000
C01859=18.500,24.775,36.587,-178.9391,1.5774,0.0000
C01860=17.826,23.134,35.561,-179.7205,-18.7836,0.0000
C01861=18.610,21.719,35.152,-158.8397,-24.0264,0.0000
C01862=19.522,20.847,35.134,-154.9228,-21.3866,0.0000
C01863=20.193,20.193,35.146,-155.7558,-22.3233,0.0000
C01864=20.846,19.522,35.134,-156.6177,-23.2450,0.0000
C01865=21.719,18.610,35.152,-154.4508,-19.2484,0.0000
C01866=23.134,17.826,35.561,-161.2167,-0.2643,0.0000
C01867=24.775,18.500,36.587,178.4223,-1.0605,0.0000
C01868=27.005,20.165,37.988,176.7172,-2.3719,0.0000
C01869=29.853,22.391,39.399,176.1159,-2.8696,0.0000
C01870=32.968,24.818,40.447,175.7483,-3.1474,0.0000
C01871=35.890,26.937,40.953,175.4165,-2.2977,0.0000
C01872=38.982,27.526,41.216,176.7723,0.3150,0.0000
C01873=41.848,26.450,41.429,178.7336,0.9130,0.0000
C01874=43.894,23.932,41.642,179.9508,0.0899,0.0000
C01875=45.474,20.785,41.781,179.9950,0.0108,0.0000
C01876=46.852,17.458,41.781,179.9959,0.0112,0.0000
C01877=47.960,14.116,41.642,179.9713,0.0983,0.0000
C01878=48.294,10.888,41.429,-179.7502,1.5410,0.0000
C01879=47.028,8.101,41.216,-177.9392,2.5046,0.0000
C01880=44.425,6.331,40.953,-175.1330,1.6109,0.0000
C01881=40.861,5.763,40.447,-174.7687,0.7747,0.0000
C01882=36.942,5.276,39.399,-175.2249,0.7127,0.0000
C01883=33.354,4.837,37.988,-176.0018,0.6414,0.0000
C01884=30.601,4.437,36.587,-178.1345,0.3654,0.0000
C01885=28.963,3.753,35.561,166.6644,-13.3530,0.0000
